					Quota_DestZ	:= Quota_PostZ + 						(* Quota Y Postazione *)
									Offset_Postazione_Z +				(* Offset Postazione *)	
									//Pallet_DimZ +						(* Dimensione/2 del Pallet/Cassa/Cavallina *)
									//Ojo formaciones en plano la altura de la base viene calculada en la  estructura
									// Forming
									Offset_Pallet_Z_90 + 				(* Offset Deposito Direzione Z del pallet *)
									Quota_FormaturaZ;					(* Quota di deposito Z da Formatura *)
										
					Quota_DestJ	:= Quota_FormaturaJ +					(* Quota di deposito Z da Formatura *)
									Offset_Pallet_J_90;					(* Offset Deposito inclinazione J del pallet *)
				
					(* Se ho l'abilitazione dell'utilizzo delle quote apprese,
						LE utilizzo come quote "buone" per eseguire il posizionamento *)				
					//Posizionamento lungo X
					//IF Apprendimento.X.Lato90.Stato = APPRENDIMENTO_ESEGUITO THEN
					//	Quota_DestX := Apprendimento.X.Lato90.QuotaRilevata;
					//END_IF
					////Posizionamento lungo Y lato 90°
					//IF Apprendimento.Y.Lato90.Stato = APPRENDIMENTO_ESEGUITO THEN
					//	Quota_DestY := Apprendimento.Y.Lato90.QuotaRilevata;
					//END_IF
					//Posizionamento lungo Z
					//Posizionamento lungo Z
					IF Apprendimento.Z.Lato90.Stato <> APPRENDIMENTO_DISABILITATO THEN
						IF Apprendimento.Z.Lato90.Stato = APPRENDIMENTO_ESEGUITO THEN
							Quota_ApproccioDestZ := Apprendimento.Z.Lato90.QuotaRilevata + Distanza_ApproccioFormaturaZ;
						ELSE
							Quota_ApproccioDestZ := Apprendimento.Z.Lato90.QuotaStart + Offset_Apprendimento_Z;
						END_IF
					ELSE
						Quota_ApproccioDestZ := Quota_DestZ +						(* Quota di deposito Z *)
												Distanza_ApproccioFormaturaZ;			(* Approccio Z da Formatura *)
					END_IF
					//Posizionamento lungo J lato 90°
					//IF Apprendimento.J.Lato90.Stato = APPRENDIMENTO_ESEGUITO THEN
					//	Quota_DestJ := Apprendimento.J.Lato90.QuotaRilevata;
					//END_IF			
				(*****************************************************************************************************************)
				(************************************************ QUOTE APPROCCIO ************************************************)
				(*****************************************************************************************************************)										
					Quota_ApproccioDestX	:= Quota_DestX;				(* Quota di deposito X *)
														
					Quota_ApproccioDestY 	:= Quota_DestY; 			(* Quota di deposito Y *)
											
					//Quota_ApproccioDestZ := Quota_DestZ +						(* Quota di deposito Z *)
					//						Distanza_ApproccioFormaturaZ;			(* Approccio Z da Formatura *)
										
					Quota_ApproccioDestJ	:= Quota_DestJ;				(* Quota di deposito J *)				
					
					
				END_IF
			{endregion}
			{Region "ANGOLO SX" }
			ANGOLO_SX :
				(*******************************************************************************************************************)
											(* Deposito su LASTRA con rotazione piano >90° e < 180°*)
				(*******************************************************************************************************************)
				IF Angolo_Destinazione > 90 THEN
					
					Quota_DestX	:= Quota_PostX + 						(* Quota X Postazione *)
									Offset_Postazione_X + 				(* Offset Postazione *)
									//Pallet_DimX/2 +						(* Dimensione/2 del Pallet/Cassa/Cavallina *)
									Offset_Pallet_X_180 +				(* Offset Deposito Direzione X del pallet *)
									Quota_FormaturaX;					(* Quota di deposito X da Formatura *)
				
					Quota_DestY := Quota_PostY + 						(* Quota Y Postazione *)
									IngombroDestinazioneY_Neg +
									Offset_Postazione_Y + 				(* Offset Postazione *)																							
									Pallet_DimY/2 +						(* Dimensione/2 del Pallet/Cassa/Cavallina *)
									Offset_Pallet_Y_180 +				(* Offset Deposito Direzione Y del pallet *)
									Quota_FormaturaY; 					(* Quota di deposito Y da Formatura *)
										
					Quota_DestZ	:= Quota_PostZ + 						(* Quota Y Postazione *)
									Offset_Postazione_Z +				(* Offset Postazione *)	
									//Pallet_DimZ +						(* Dimensione/2 del Pallet/Cassa/Cavallina *)
									Offset_Pallet_Z_180 + 				(* Offset Deposito Direzione Z del pallet *)
									(-ScostamentoVerticalePuntoCentrale) +		(* Sporgenza rispetto al filo pinza quando è in orizzontale *)
									Quota_FormaturaZ;					(* Quota di deposito Z da Formatura *)
							
					Quota_DestJ	:= Quota_FormaturaJ +					(* Quota di deposito Z da Formatura *)
									Offset_Pallet_J_180;				(* Offset Deposito inclinazione J del pallet *)
									
					(* Se ho l'abilitazione dell'utilizzo delle quote apprese,
						LE utilizzo come quote "buone" per eseguire il posizionamento *)				
					//Posizionamento lungo X
					IF Apprendimento.X.Lato180.Stato = APPRENDIMENTO_ESEGUITO THEN
						Quota_DestX := Apprendimento.X.Lato180.QuotaRilevata;
					END_IF
					//Posizionamento lungo Y lato 180°
					IF Apprendimento.Y.Lato180.Stato = APPRENDIMENTO_ESEGUITO THEN
						Quota_DestY := Apprendimento.Y.Lato180.QuotaRilevata;
					END_IF
					//Posizionamento lungo Z
					IF Apprendimento.Z.Lato180.Stato = APPRENDIMENTO_ESEGUITO THEN
						Quota_DestZ := Apprendimento.Z.Lato180.QuotaRilevata;
					END_IF
					//Posizionamento lungo J lato 180°
					IF Apprendimento.J.Lato180.Stato = APPRENDIMENTO_ESEGUITO THEN
						Quota_DestJ := Apprendimento.J.Lato180.QuotaRilevata;
					END_IF
				(*****************************************************************************************************************)
				(************************************************ QUOTE APPROCCIO ************************************************)
				(*****************************************************************************************************************)	
					
					(* Valutazione della Direzione dell'Asse X*)
					IF PosizioneAttuale_X >= Quota_DestX THEN // La posizione attuale è maggiore della posizione di destinazione 
						Quota_ApproccioDestX := Quota_DestX +					(* Quota di deposito X *)
												Distanza_ApproccioFormaturaX;		(* Approccio X da Formatura *)	
					ELSE // La posizione attuale è minore della posizione di destinazione 
						Quota_ApproccioDestX := Quota_DestX -					(* Quota di deposito X *)
												Distanza_ApproccioFormaturaX;		(* Approccio X da Formatura *)
					END_IF			
				
					Quota_ApproccioDestY := Quota_DestY + 						(* Quota di deposito Y *)
											Distanza_ApproccioFormaturaY; 			(* Approccio Y da Formatura *)
										
					Quota_ApproccioDestZ := Quota_DestZ +						(* Quota di deposito Z da Formatura *)
											Distanza_ApproccioFormaturaZ;			(* Approccio Z da Formatura *)
							
					Quota_ApproccioDestJ := Quota_DestJ +						(* Quota di deposito J da Forma*)	
											Distanza_ApproccioFormaturaJ;			(* Approccio J da Formatura *)
				(*******************************************************************************************************************)						
											(* Deposito su LASTRA con rotazione piano < 90° e >0°*)	
				(*******************************************************************************************************************)							
				ELSIF Angolo_Destinazione < 90 THEN
					
					Quota_DestX	:= Quota_PostX + 						(* Quota X Postazione *)
									Offset_Postazione_X + 				(* Offset Postazione *)
									//Pallet_DimX/2 +						(* Dimensione/2 del Pallet/Cassa/Cavallina *)
									Offset_Pallet_X_0 +					(* Offset Deposito Direzione X del pallet *)
									Quota_FormaturaX;					(* Quota di deposito X da Formatura *)
				
					Quota_DestY := Quota_PostY - 						(* Quota Y Postazione *)
									IngombroDestinazioneY_Pos +
									Offset_Postazione_Y + 				(* Offset Postazione *)																								
									Pallet_DimY/2 +						(* Dimensione/2 del Pallet/Cassa/Cavallina *)
									Offset_Pallet_Y_0 -					(* Offset Deposito Direzione Y del pallet *)
									Quota_FormaturaY; 					(* Quota di deposito Y da Formatura *)
										
					Quota_DestZ	:= Quota_PostZ + 						(* Quota Y Postazione *)
									Offset_Postazione_Z +				(* Offset Postazione *)	
									//Pallet_DimZ +						(* Dimensione/2 del Pallet/Cassa/Cavallina *)
									Offset_Pallet_Z_0 + 				(* Offset Deposito Direzione Z del pallet *)
									(-ScostamentoVerticalePuntoCentrale) +		(* Sporgenza rispetto al filo pinza quando è in orizzontale *)
									Quota_FormaturaZ;					(* Quota di deposito Z da Formatura *)
							
					Quota_DestJ	:= Quota_FormaturaJ +					(* Quota di deposito Z da Formatura *)
									Offset_Pallet_J_0;					(* Offset Deposito inclinazione J del pallet *)
									
					(* Se ho l'abilitazione dell'utilizzo delle quote apprese,
						LE utilizzo come quote "buone" per eseguire il posizionamento *)				
					//Posizionamento lungo X
					IF Apprendimento.X.Lato0.Stato = APPRENDIMENTO_ESEGUITO THEN
						Quota_DestX := Apprendimento.X.Lato0.QuotaRilevata;
					END_IF
					//Posizionamento lungo Y lato 0°
					IF Apprendimento.Y.Lato0.Stato = APPRENDIMENTO_ESEGUITO THEN
						Quota_DestY := Apprendimento.Y.Lato0.QuotaRilevata;
					END_IF
					//Posizionamento lungo Z
					IF Apprendimento.Z.Lato0.Stato = APPRENDIMENTO_ESEGUITO THEN
						Quota_DestZ := Apprendimento.Z.Lato0.QuotaRilevata;
					END_IF
					//Posizionamento lungo J lato 0°
					IF Apprendimento.J.Lato0.Stato = APPRENDIMENTO_ESEGUITO THEN
						Quota_DestJ := Apprendimento.J.Lato0.QuotaRilevata;
					END_IF
				(*****************************************************************************************************************)
				(************************************************ QUOTE APPROCCIO ************************************************)
				(*****************************************************************************************************************)	
					
					(* Valutazione della Direzione dell'Asse X*)
					IF PosizioneAttuale_X >= Quota_DestX THEN // La posizione attuale è maggiore della posizione di destinazione 
						Quota_ApproccioDestX := Quota_DestX +					(* Quota di deposito X *)
												Distanza_ApproccioFormaturaX;		(* Approccio X da Formatura *)	
					ELSE // La posizione attuale è minore della posizione di destinazione 
						Quota_ApproccioDestX := Quota_DestX -					(* Quota di deposito X *)
												Distanza_ApproccioFormaturaX;		(* Approccio X da Formatura *)
					END_IF			
				
					Quota_ApproccioDestY := Quota_DestY - 						(* Quota di deposito Y *)
											Distanza_ApproccioFormaturaY; 			(* Approccio Y da Formatura *)
										
					Quota_ApproccioDestZ := Quota_DestZ +						(* Quota di deposito Z *)
											Distanza_ApproccioFormaturaZ;			(* Approccio Z da Formatura *)
							
					Quota_ApproccioDestJ := Quota_DestJ +						(* Quota di deposito J *)
											Distanza_ApproccioFormaturaJ;			(* Approccio J da Formatura *)
							
				(*******************************************************************************************************************)						
											(* Deposito su LASTRA in cassa con rotazione piano = 90° *)
				(*******************************************************************************************************************)
				ELSE
					
					Quota_DestX	:= Quota_PostX + 						(* Quota X Postazione *)
									Offset_Postazione_X + 				(* Offset Postazione *)
									Pallet_DimX/2 +						(* Dimensione/2 del Pallet/Cassa/Cavallina *)
									Offset_Pallet_X_90;// +				(* Offset Deposito Direzione X del pallet *)
									//Quota_FormaturaX;					(* Quota di deposito X da Formatura *)
										
					Quota_DestY := Quota_PostY + 						(* Quota Y Postazione *)
									Offset_Postazione_Y + 				(* Offset Postazione *)																							
									Pallet_DimY/2 +						(* Dimensione/2 del Pallet/Cassa/Cavallina *)
									Offset_Pallet_Y_90;// +				(* Offset Deposito Direzione Y del pallet *)
									//Quota_FormaturaY; 					(* Quota di deposito Y da Formatura *)
											
					Quota_DestZ	:= Quota_PostZ + 						(* Quota Y Postazione *)
									Offset_Postazione_Z +				(* Offset Postazione *)	
									//Pallet_DimZ +						(* Dimensione/2 del Pallet/Cassa/Cavallina *)
									Offset_Pallet_Z_90 + 				(* Offset Deposito Direzione Z del pallet *)
									Quota_FormaturaZ;					(* Quota di deposito Z da Formatura *)
										
					Quota_DestJ	:= Quota_FormaturaJ;// +					(* Quota di deposito Z da Formatura *)
									//Offset_Pallet_J_90;					(* Offset Deposito inclinazione J del pallet *)
									
					(* Se ho l'abilitazione dell'utilizzo delle quote apprese,
						LE utilizzo come quote "buone" per eseguire il posizionamento *)				
					//Posizionamento lungo X
					IF Apprendimento.X.Lato90.Stato = APPRENDIMENTO_ESEGUITO THEN
						Quota_DestX := Apprendimento.X.Lato90.QuotaRilevata;
					END_IF
					//Posizionamento lungo Y lato 90°
					IF Apprendimento.Y.Lato90.Stato = APPRENDIMENTO_ESEGUITO THEN
						Quota_DestY := Apprendimento.Y.Lato90.QuotaRilevata;
					END_IF
					//Posizionamento lungo Z
					//IF Apprendimento.Z.Lato90.Stato = APPRENDIMENTO_ESEGUITO THEN
					//	Quota_DestZ := Apprendimento.Z.Lato90.QuotaRilevata + Offset_Apprendimento_Z;
					//ELSE
					//	Quota_DestZ := Apprendimento.Z.Lato90.QuotaStart;
					//END_IF
					//Posizionamento lungo Z
					IF Apprendimento.Z.Lato90.Stato <> APPRENDIMENTO_DISABILITATO THEN
						IF Apprendimento.Z.Lato90.Stato = APPRENDIMENTO_ESEGUITO THEN
							Quota_ApproccioDestZ := Apprendimento.Z.Lato90.QuotaRilevata + Distanza_ApproccioFormaturaZ;
						ELSE
							Quota_ApproccioDestZ := Apprendimento.Z.Lato90.QuotaStart + Offset_Apprendimento_Z;
						END_IF
					ELSE
						Quota_ApproccioDestZ := Quota_DestZ +						(* Quota di deposito Z *)
												Distanza_ApproccioFormaturaZ;			(* Approccio Z da Formatura *)
					END_IF		  
										
					//Posizionamento lungo J lato 90°
					IF Apprendimento.J.Lato90.Stato = APPRENDIMENTO_ESEGUITO THEN
						Quota_DestJ := Apprendimento.J.Lato90.QuotaRilevata;
					END_IF
							
				(*****************************************************************************************************************)
				(************************************************ QUOTE APPROCCIO ************************************************)
				(*****************************************************************************************************************)										
					Quota_ApproccioDestX	:= Quota_DestX;				(* Quota di deposito X *)
														
					Quota_ApproccioDestY 	:= Quota_DestY; 			(* Quota di deposito Y *)
											
					////Quota_ApproccioDestZ := Quota_DestZ +						(* Quota di deposito Z *)
					//						Distanza_ApproccioFormaturaZ;			(* Approccio Z da Formatura *)
										
					Quota_ApproccioDestJ	:= Quota_DestJ;				(* Quota di deposito J *)				
					
				END_IF
			{endregion}
			{Region "XDX_YCENTRALE" }
			XDX_YCENTRALE:
				(*******************************************************************************************************************)
											(* Deposito su LASTRA con rotazione piano >90° e < 180°*)
				(*******************************************************************************************************************)																		
				IF Angolo_Destinazione > 90 THEN
					
					Quota_DestX	:= Quota_PostX + 						(* Quota X Postazione *)
									Offset_Postazione_X - 				(* Offset Postazione *)
									Pallet_DimX/2 +						(* Dimensione/2 del Pallet/Cassa/Cavallina *)
									Offset_Pallet_X_180 +				(* Offset Deposito Direzione X del pallet *)
									Quota_FormaturaX;					(* Quota di deposito X da Formatura *)
				
					Quota_DestY := Quota_PostY + 						(* Quota Y Postazione *)
									Offset_Postazione_Y + 				(* Offset Postazione *)																								
									Pallet_DimY/2 -						(* Dimensione/2 del Pallet/Cassa/Cavallina *)
									//Offset_Pallet_Y_180 +				(* Offset Deposito Direzione Y del pallet *)
									Quota_FormaturaY; 					(* Quota di deposito Y da Formatura *)
										
					Quota_DestZ	:= Quota_PostZ + 						(* Quota Y Postazione *)
									Offset_Postazione_Z +				(* Offset Postazione *)	
									Pallet_DimZ +						(* Dimensione/2 del Pallet/Cassa/Cavallina *)
									Offset_Pallet_Z_180 + 				(* Offset Deposito Direzione Z del pallet *)
									Quota_FormaturaZ;					(* Quota di deposito Z da Formatura *)
							
					Quota_DestJ	:= Quota_FormaturaJ +					(* Quota di deposito Z da Formatura *)
									Offset_Pallet_J_180;				(* Offset Deposito inclinazione J del pallet *)
									
					(* Se ho l'abilitazione dell'utilizzo delle quote apprese,
						LE utilizzo come quote "buone" per eseguire il posizionamento *)				
					//Posizionamento lungo X
					IF Apprendimento.X.Lato180.Stato = APPRENDIMENTO_ESEGUITO THEN
						Quota_DestX := Apprendimento.X.Lato180.QuotaRilevata;
					END_IF
					//Posizionamento lungo Y lato 180°
					//IF Apprendimento.Y.Lato180.Stato = APPRENDIMENTO_ESEGUITO THEN
					//	Quota_DestY := Apprendimento.Y.Lato180.QuotaRilevata;
					//END_IF
					//Posizionamento lungo Z
					IF Apprendimento.Z.Lato180.Stato = APPRENDIMENTO_ESEGUITO THEN
						Quota_DestZ := Apprendimento.Z.Lato180.QuotaRilevata;
					END_IF
					//Posizionamento lungo J lato 180°
					IF Apprendimento.J.Lato180.Stato = APPRENDIMENTO_ESEGUITO THEN
						Quota_DestJ := Apprendimento.J.Lato180.QuotaRilevata;
					END_IF
									
				(*****************************************************************************************************************)
				(************************************************ QUOTE APPROCCIO ************************************************)
				(*****************************************************************************************************************)	
					Quota_ApproccioDestX	:= Quota_DestX;				(* Quota di deposito X *)
					//Quota_ApproccioDestY 	:= Quota_DestY; 			(* Quota di deposito Y *)
					IF CicloDiPrelievo THEN
						IF Apprendimento.Y.Lato90.Stato = APPRENDIMENTO_ESEGUITO THEN
							Quota_ApproccioDestY := Apprendimento.Y.Lato90.QuotaRilevata +	(* Quota rilevata Z *)
													Distanza_ApproccioFormaturaY;			(* Approccio Z da Formatura *)				
						ELSIF Apprendimento.Y.Lato90.Stato <> APPRENDIMENTO_ESEGUITO THEN
							Quota_ApproccioDestY := Quota_DestY + 						(* Quota di deposito Y *)
													Distanza_ApproccioFormaturaY+ 			(* Approccio Y da Formatura *)
													Offset_Apprendimento_Y;							
						END_IF
					ELSE
						//Posizionamento lungo Z lato 90°
						IF Apprendimento.Y.Lato90.Stato = APPRENDIMENTO_ESEGUITO THEN
							Quota_DestY := Apprendimento.Y.Lato90.QuotaRilevata +
											Distanza_ApproccioFormaturaY;
						END_IF
					END_IF
					
					Quota_ApproccioDestZ := Quota_DestZ +						(* Quota di deposito Z *)
											Distanza_ApproccioFormaturaZ;			(* Approccio Z da Formatura *)
										
					Quota_ApproccioDestJ	:= Quota_DestJ;				(* Quota di deposito J *)				
									
				(*******************************************************************************************************************)						
											(* Deposito su LASTRA con rotazione piano < 90° e >0°*)	
				(*******************************************************************************************************************)							
				ELSIF Angolo_Destinazione < 90 THEN
					
					Quota_DestX	:= Quota_PostX + 						(* Quota X Postazione *)
									Offset_Postazione_X - 				(* Offset Postazione *)
									Pallet_DimX/2 +						(* Dimensione/2 del Pallet/Cassa/Cavallina *)
									Offset_Pallet_X_0 +					(* Offset Deposito Direzione X del pallet *)
									Quota_FormaturaX;					(* Quota di deposito X da Formatura *)
				
					Quota_DestY := Quota_PostY - 						(* Quota Y Postazione *)
									Offset_Postazione_Y - 				(* Offset Postazione *)																							
									Pallet_DimY/2 -						(* Dimensione/2 del Pallet/Cassa/Cavallina *)
									//Offset_Pallet_Y_0 +					(* Offset Deposito Direzione Y del pallet *)
									Quota_FormaturaY; 					(* Quota di deposito Y da Formatura *)
										
					Quota_DestZ	:= Quota_PostZ + 						(* Quota Y Postazione *)
									Offset_Postazione_Z +				(* Offset Postazione *)	
									Pallet_DimZ +						(* Dimensione/2 del Pallet/Cassa/Cavallina *)
									Offset_Pallet_Z_0 + 				(* Offset Deposito Direzione Z del pallet *)
									Quota_FormaturaZ;					(* Quota di deposito Z da Formatura *)
							
					Quota_DestJ	:= Quota_FormaturaJ +					(* Quota di deposito Z da Formatura *)
									Offset_Pallet_J_0;					(* Offset Deposito inclinazione J del pallet *)
									
					(* Se ho l'abilitazione dell'utilizzo delle quote apprese,
						LE utilizzo come quote "buone" per eseguire il posizionamento *)				
					//Posizionamento lungo X
					IF Apprendimento.X.Lato0.Stato = APPRENDIMENTO_ESEGUITO THEN
						Quota_DestX := Apprendimento.X.Lato0.QuotaRilevata;
					END_IF
					//Posizionamento lungo Y lato 0°
					//IF Apprendimento.Y.Lato0.Stato = APPRENDIMENTO_ESEGUITO THEN
					//	Quota_DestY := Apprendimento.Y.Lato0.QuotaRilevata;
					//END_IF
					IF CicloDiPrelievo THEN
						IF Apprendimento.Y.Lato90.Stato = APPRENDIMENTO_ESEGUITO THEN
							Quota_ApproccioDestY := Apprendimento.Y.Lato90.QuotaRilevata -	(* Quota rilevata Z *)
													Distanza_ApproccioFormaturaY;			(* Approccio Z da Formatura *)				
						ELSIF Apprendimento.Y.Lato90.Stato <> APPRENDIMENTO_ESEGUITO THEN
							Quota_ApproccioDestY := Quota_DestY - 						(* Quota di deposito Y *)
													Distanza_ApproccioFormaturaY- 			(* Approccio Y da Formatura *)
													Offset_Apprendimento_Y;							
						END_IF
					ELSE
						//Posizionamento lungo Z lato 90°
						IF Apprendimento.Y.Lato90.Stato = APPRENDIMENTO_ESEGUITO THEN
							Quota_DestY := Apprendimento.Y.Lato90.QuotaRilevata -
											Distanza_ApproccioFormaturaY;
						END_IF
					END_IF
					//Posizionamento lungo Z
					IF Apprendimento.Z.Lato0.Stato = APPRENDIMENTO_ESEGUITO THEN
						Quota_DestZ := Apprendimento.Z.Lato0.QuotaRilevata;
					END_IF
					//Posizionamento lungo J lato 0°
					IF Apprendimento.J.Lato0.Stato = APPRENDIMENTO_ESEGUITO THEN
						Quota_DestJ := Apprendimento.J.Lato0.QuotaRilevata;
					END_IF
									
				(*****************************************************************************************************************)
				(************************************************ QUOTE APPROCCIO ************************************************)
				(*****************************************************************************************************************)	
					
					(* Valutazione della Direzione dell'Asse X*)
					IF PosizioneAttuale_X >= Quota_DestX THEN // La posizione attuale è maggiore della posizione di destinazione 
						Quota_ApproccioDestX := Quota_DestX +					(* Quota di deposito X *)
												Distanza_ApproccioFormaturaX;		(* Approccio X da Formatura *)	
					ELSE // La posizione attuale è minore della posizione di destinazione 
						Quota_ApproccioDestX := Quota_DestX -					(* Quota di deposito X *)
												Distanza_ApproccioFormaturaX;		(* Approccio X da Formatura *)
					END_IF			
				
					Quota_ApproccioDestY := Quota_DestY - 						(* Quota di deposito Y *)
											Distanza_ApproccioFormaturaY; 			(* Approccio Y da Formatura *)
										
					Quota_ApproccioDestZ := Quota_DestZ +						(* Quota di deposito Z *)
											Distanza_ApproccioFormaturaZ;			(* Approccio Z da Formatura *)
							
					Quota_ApproccioDestJ := Quota_DestJ +						(* Quota di deposito J *)
											Distanza_ApproccioFormaturaJ;			(* Approccio J da Formatura *)				
							
				(*******************************************************************************************************************)						
											(* Deposito su LASTRA in cassa con rotazione piano = 90° *)
				(*******************************************************************************************************************)
				ELSE
					
					Quota_DestX	:= Quota_PostX + 						(* Quota X Postazione *)
									Offset_Postazione_X - 				(* Offset Postazione *)
									Pallet_DimX/2 +						(* Dimensione/2 del Pallet/Cassa/Cavallina *)
									Offset_Pallet_X_90 +				(* Offset Deposito Direzione X del pallet *)
									Quota_FormaturaX;					(* Quota di deposito X da Formatura *)
														
					Quota_DestY := Quota_PostY + 						(* Quota Y Postazione *)
									Offset_Postazione_Y + 				(* Offset Postazione *)																							
									//Pallet_DimY/2 +						(* Dimensione/2 del Pallet/Cassa/Cavallina *)
									//Offset_Pallet_Y_90 +				(* Offset Deposito Direzione Y del pallet *)
									Quota_FormaturaY; 					(* Quota di deposito Y da Formatura *)
											
					Quota_DestZ	:= Quota_PostZ + 						(* Quota Y Postazione *)
									Offset_Postazione_Z +				(* Offset Postazione *)	
									Pallet_DimZ +						(* Dimensione/2 del Pallet/Cassa/Cavallina *)
									Offset_Pallet_Z_90 + 				(* Offset Deposito Direzione Z del pallet *)
									Quota_FormaturaZ;					(* Quota di deposito Z da Formatura *)
										
					Quota_DestJ	:= Quota_FormaturaJ +					(* Quota di deposito Z da Formatura *)
									Offset_Pallet_J_90;					(* Offset Deposito inclinazione J del pallet *)
					
					(* Se ho l'abilitazione dell'utilizzo delle quote apprese,
						LE utilizzo come quote "buone" per eseguire il posizionamento *)				
					//Posizionamento lungo X
					IF Apprendimento.X.Lato90.Stato = APPRENDIMENTO_ESEGUITO THEN
						Quota_DestX := Apprendimento.X.Lato90.QuotaRilevata;
					END_IF
					//Posizionamento lungo Y lato 90°
					IF Apprendimento.Y.Lato90.Stato = APPRENDIMENTO_ESEGUITO THEN
						Quota_DestY := Apprendimento.Y.Lato90.QuotaRilevata;
					END_IF
					//Posizionamento lungo Z
					IF CicloDiPrelievo THEN
						IF Apprendimento.Z.Lato90.Stato = APPRENDIMENTO_ESEGUITO THEN
							Quota_ApproccioDestZ := Apprendimento.Z.Lato90.QuotaRilevata +	(* Quota rilevata Z *)
													Distanza_ApproccioFormaturaZ;			(* Approccio Z da Formatura *)				
						ELSIF Apprendimento.Z.Lato90.Stato <> APPRENDIMENTO_ESEGUITO THEN
							Quota_ApproccioDestZ := Quota_PostZ + 						(* Quota Y Postazione *)
													Offset_Postazione_Z +				(* Offset Postazione *)	
													Offset_Pallet_Z_0 +					(* Offset Direzione Z del pall*)
													HmaxElemento +						(* Quota di deposito Z *)
													Offset_Apprendimento_Z;							
						END_IF
					ELSE
						//Posizionamento lungo Z lato 90°
						IF Apprendimento.Z.Lato90.Stato = APPRENDIMENTO_ESEGUITO THEN
							Quota_DestZ := Apprendimento.Z.Lato90.QuotaRilevata;
						END_IF
						Quota_ApproccioDestZ := Quota_DestZ +						(* Quota di deposito Z *)
												Distanza_ApproccioFormaturaZ;			(* Approccio Z da Formatura *)
					END_IF
					//Posizionamento lungo J lato 90°
					IF Apprendimento.J.Lato90.Stato = APPRENDIMENTO_ESEGUITO THEN
						Quota_DestJ := Apprendimento.J.Lato90.QuotaRilevata;
					END_IF
									
				(*****************************************************************************************************************)
				(************************************************ QUOTE APPROCCIO ************************************************)
				(*****************************************************************************************************************)										
					Quota_ApproccioDestX	:= Quota_DestX;				(* Quota di deposito X *)
														
					Quota_ApproccioDestY 	:= Quota_DestY; 			(* Quota di deposito Y *)
											
					//Quota_ApproccioDestZ := Quota_DestZ +						(* Quota di deposito Z *)
					//						Distanza_ApproccioFormaturaZ;			(* Approccio Z da Formatura *)
										
					Quota_ApproccioDestJ	:= Quota_DestJ;				(* Quota di deposito J *)				
				END_IF
			{endregion}
			{Region "XSX_YCENTRALE" }
			XSX_YCENTRALE:
				(*******************************************************************************************************************)
											(* Deposito su LASTRA con rotazione piano >90° e < 180°*)
				(*******************************************************************************************************************)
				IF Angolo_Destinazione > 90 THEN
					
					Quota_DestX	:= Quota_PostX + 						(* Quota X Postazione *)
									Offset_Postazione_X + 				(* Offset Postazione *)
									Pallet_DimX/2 +						(* Dimensione/2 del Pallet/Cassa/Cavallina *)
									Offset_Pallet_X_180 +				(* Offset Deposito Direzione X del pallet *)
									Quota_FormaturaX;					(* Quota di deposito X da Formatura *)
				
					Quota_DestY := Quota_PostY + 						(* Quota Y Postazione *)
									Offset_Postazione_Y + 				(* Offset Postazione *)																							
									//Pallet_DimY/2 +						(* Dimensione/2 del Pallet/Cassa/Cavallina *)
									//Offset_Pallet_Y_180 +				(* Offset Deposito Direzione Y del pallet *)
									Quota_FormaturaY; 					(* Quota di deposito Y da Formatura *)
										
					Quota_DestZ	:= Quota_PostZ + 						(* Quota Y Postazione *)
									Offset_Postazione_Z +				(* Offset Postazione *)	
									Pallet_DimZ +						(* Dimensione/2 del Pallet/Cassa/Cavallina *)
									Offset_Pallet_Z_180 + 				(* Offset Deposito Direzione Z del pallet *)
									Quota_FormaturaZ;					(* Quota di deposito Z da Formatura *)
							
					Quota_DestJ	:= Quota_FormaturaJ +					(* Quota di deposito Z da Formatura *)
									Offset_Pallet_J_180;				(* Offset Deposito inclinazione J del pallet *)
									
					(* Se ho l'abilitazione dell'utilizzo delle quote apprese,
						LE utilizzo come quote "buone" per eseguire il posizionamento *)				
					//Posizionamento lungo X
					IF Apprendimento.X.Lato180.Stato = APPRENDIMENTO_ESEGUITO THEN
						Quota_DestX := Apprendimento.X.Lato180.QuotaRilevata;
					END_IF
					//Posizionamento lungo Y lato 180°
					IF Apprendimento.Y.Lato180.Stato = APPRENDIMENTO_ESEGUITO THEN
						Quota_DestY := Apprendimento.Y.Lato180.QuotaRilevata;
					END_IF
					//Posizionamento lungo Z
					IF Apprendimento.Z.Lato180.Stato = APPRENDIMENTO_ESEGUITO THEN
						Quota_DestZ := Apprendimento.Z.Lato180.QuotaRilevata;
					END_IF
					//Posizionamento lungo J lato 180°
					IF Apprendimento.J.Lato180.Stato = APPRENDIMENTO_ESEGUITO THEN
						Quota_DestJ := Apprendimento.J.Lato180.QuotaRilevata;
					END_IF				
					
				(*****************************************************************************************************************)
				(************************************************ QUOTE APPROCCIO ************************************************)
				(*****************************************************************************************************************)	
					
					(* Valutazione della Direzione dell'Asse X*)
					IF PosizioneAttuale_X >= Quota_DestX THEN // La posizione attuale è maggiore della posizione di destinazione 
						Quota_ApproccioDestX := Quota_DestX +					(* Quota di deposito X *)
												Distanza_ApproccioFormaturaX;		(* Approccio X da Formatura *)	
					ELSE // La posizione attuale è minore della posizione di destinazione 
						Quota_ApproccioDestX := Quota_DestX -					(* Quota di deposito X *)
												Distanza_ApproccioFormaturaX;		(* Approccio X da Formatura *)
					END_IF			
				
					Quota_ApproccioDestY := Quota_DestY + 						(* Quota di deposito Y *)
											Distanza_ApproccioFormaturaY; 			(* Approccio Y da Formatura *)
										
					Quota_ApproccioDestZ := Quota_DestZ +						(* Quota di deposito Z da Formatura *)
											Distanza_ApproccioFormaturaZ;			(* Approccio Z da Formatura *)
							
					Quota_ApproccioDestJ := Quota_DestJ +						(* Quota di deposito J da Forma*)	
											Distanza_ApproccioFormaturaJ;			(* Approccio J da Formatura *)
				(*******************************************************************************************************************)						
											(* Deposito su LASTRA con rotazione piano < 90° e >0°*)	
				(*******************************************************************************************************************)							
				ELSIF Angolo_Destinazione < 90 THEN
					
					Quota_DestX	:= Quota_PostX + 						(* Quota X Postazione *)
									Offset_Postazione_X + 				(* Offset Postazione *)
									Pallet_DimX/2 +						(* Dimensione/2 del Pallet/Cassa/Cavallina *)
									Offset_Pallet_X_0 +					(* Offset Deposito Direzione X del pallet *)
									Quota_FormaturaX;					(* Quota di deposito X da Formatura *)
				
					Quota_DestY := Quota_PostY + 						(* Quota Y Postazione *)
									Offset_Postazione_Y + 				(* Offset Postazione *)																								
									//Pallet_DimY/2 -						(* Dimensione/2 del Pallet/Cassa/Cavallina *)
									//Offset_Pallet_Y_0 +					(* Offset Deposito Direzione Y del pallet *)
									Quota_FormaturaY; 					(* Quota di deposito Y da Formatura *)
										
					Quota_DestZ	:= Quota_PostZ + 						(* Quota Y Postazione *)
									Offset_Postazione_Z +				(* Offset Postazione *)	
									Pallet_DimZ +						(* Dimensione/2 del Pallet/Cassa/Cavallina *)
									Offset_Pallet_Z_90 + 				(* Offset Deposito Direzione Z del pallet *)
									Quota_FormaturaZ;					(* Quota di deposito Z da Formatura *)
							
					Quota_DestJ	:= Quota_FormaturaJ +					(* Quota di deposito Z da Formatura *)
									Offset_Pallet_J_0;					(* Offset Deposito inclinazione J del pallet *)
									
					(* Se ho l'abilitazione dell'utilizzo delle quote apprese,
						LE utilizzo come quote "buone" per eseguire il posizionamento *)				
					//Posizionamento lungo X
					IF Apprendimento.X.Lato0.Stato = APPRENDIMENTO_ESEGUITO THEN
						Quota_DestX := Apprendimento.X.Lato0.QuotaRilevata;
					END_IF
					//Posizionamento lungo Y lato 0°
					IF Apprendimento.Y.Lato0.Stato = APPRENDIMENTO_ESEGUITO THEN
						Quota_DestY := Apprendimento.Y.Lato0.QuotaRilevata;
					END_IF
					//Posizionamento lungo Z
					IF Apprendimento.Z.Lato0.Stato = APPRENDIMENTO_ESEGUITO THEN
						Quota_DestZ := Apprendimento.Z.Lato0.QuotaRilevata;
					END_IF
					//Posizionamento lungo J lato 0°
					IF Apprendimento.J.Lato0.Stato = APPRENDIMENTO_ESEGUITO THEN
						Quota_DestJ := Apprendimento.J.Lato0.QuotaRilevata;
					END_IF		
					
				(*****************************************************************************************************************)
				(************************************************ QUOTE APPROCCIO ************************************************)
				(*****************************************************************************************************************)	
					
					(* Valutazione della Direzione dell'Asse X*)
					IF PosizioneAttuale_X >= Quota_DestX THEN // La posizione attuale è maggiore della posizione di destinazione 
						Quota_ApproccioDestX := Quota_DestX +					(* Quota di deposito X *)
												Distanza_ApproccioFormaturaX;		(* Approccio X da Formatura *)	
					ELSE // La posizione attuale è minore della posizione di destinazione 
						Quota_ApproccioDestX := Quota_DestX -					(* Quota di deposito X *)
												Distanza_ApproccioFormaturaX;		(* Approccio X da Formatura *)
					END_IF			
				
					Quota_ApproccioDestY := Quota_DestY - 						(* Quota di deposito Y *)
											Distanza_ApproccioFormaturaY; 			(* Approccio Y da Formatura *)
										
					Quota_ApproccioDestZ := Quota_DestZ +						(* Quota di deposito Z *)
											Distanza_ApproccioFormaturaZ;			(* Approccio Z da Formatura *)
							
					Quota_ApproccioDestJ := Quota_DestJ +						(* Quota di deposito J *)
											Distanza_ApproccioFormaturaJ;			(* Approccio J da Formatura *)
							
				(*******************************************************************************************************************)						
											(* Deposito su LASTRA in cassa con rotazione piano = 90° *)
				(*******************************************************************************************************************)
				ELSE
					
					Quota_DestX	:= Quota_PostX + 						(* Quota X Postazione *)
									Offset_Postazione_X + 				(* Offset Postazione *)
									Pallet_DimX/2 +						(* Dimensione/2 del Pallet/Cassa/Cavallina *)
									Offset_Pallet_X_90 +				(* Offset Deposito Direzione X del pallet *)
									Quota_FormaturaX;					(* Quota di deposito X da Formatura *)
										
					Quota_DestY := Quota_PostY + 						(* Quota Y Postazione *)
									Offset_Postazione_Y + 				(* Offset Postazione *)																							
									//Pallet_DimY/2 +						(* Dimensione/2 del Pallet/Cassa/Cavallina *)
									//Offset_Pallet_Y_90 +				(* Offset Deposito Direzione Y del pallet *)
									Quota_FormaturaY; 					(* Quota di deposito Y da Formatura *)
											
					Quota_DestZ	:= Quota_PostZ + 						(* Quota Y Postazione *)
									Offset_Postazione_Z +				(* Offset Postazione *)	
									Pallet_DimZ +						(* Dimensione/2 del Pallet/Cassa/Cavallina *)
									Offset_Pallet_Z_90 + 				(* Offset Deposito Direzione Z del pallet *)
									Quota_FormaturaZ;					(* Quota di deposito Z da Formatura *)
										
					Quota_DestJ	:= Quota_FormaturaJ +					(* Quota di deposito Z da Formatura *)
									Offset_Pallet_J_90;					(* Offset Deposito inclinazione J del pallet *)
					
					(* Se ho l'abilitazione dell'utilizzo delle quote apprese,
						LE utilizzo come quote "buone" per eseguire il posizionamento *)				
					//Posizionamento lungo X
					IF Apprendimento.X.Lato0.Stato = APPRENDIMENTO_ESEGUITO THEN
						Quota_DestX := Apprendimento.X.Lato0.QuotaRilevata;
					END_IF
					//Posizionamento lungo Y lato 0°
					IF Apprendimento.Y.Lato0.Stato = APPRENDIMENTO_ESEGUITO THEN
						Quota_DestY := Apprendimento.Y.Lato0.QuotaRilevata;
					END_IF
					//Posizionamento lungo Z
					IF Apprendimento.Z.Lato0.Stato = APPRENDIMENTO_ESEGUITO THEN
						Quota_DestZ := Apprendimento.Z.Lato0.QuotaRilevata;
					END_IF
					//Posizionamento lungo J lato 0°
					IF Apprendimento.J.Lato0.Stato = APPRENDIMENTO_ESEGUITO THEN
						Quota_DestJ := Apprendimento.J.Lato0.QuotaRilevata;
					END_IF	
				(*****************************************************************************************************************)
				(************************************************ QUOTE APPROCCIO ************************************************)
				(*****************************************************************************************************************)										
					Quota_ApproccioDestX	:= Quota_DestX;				(* Quota di deposito X *)
														
					Quota_ApproccioDestY 	:= Quota_DestY; 			(* Quota di deposito Y *)
											
					Quota_ApproccioDestZ := Quota_DestZ +						(* Quota di deposito Z *)
											Distanza_ApproccioFormaturaZ;			(* Approccio Z da Formatura *)
										
					Quota_ApproccioDestJ	:= Quota_DestJ;				(* Quota di deposito J *)
					
				END_IF
			{endregion}		
							
		ELSE
			Errore.Code := ErrWAM_FTC_PostazioneNONDefinita;
		END_CASE
	{endregion}	
	ELSE
		Errore.Code := ErrGENERICO;		
END_CASE
{region " Gestione Approccio "}	
CASE TipologiaTraiettoria OF
	
	TRAIETTORIA_CON_APPROCCIO:
		RETURN;
	
	TRAIETTORIA_SENZA_APPROCCIO:
		(*****************************************************************************************************************)
		(************************************************ QUOTE APPROCCIO ************************************************)
		(*****************************************************************************************************************)										
		Quota_ApproccioDestX	:= Quota_DestX;				(* Quota di deposito X *)
											
		Quota_ApproccioDestY 	:= Quota_DestY; 			(* Quota di deposito Y *)
								
		Quota_ApproccioDestZ 	:= Quota_DestZ; 			(* Quota di deposito Z *)
							
		Quota_ApproccioDestJ	:= Quota_DestJ;				(* Quota di deposito J *)
		RETURN;	
END_CASE
{endregion}

END_FUNCTION_BLOCK

// ---- POUs/TFPalletizerData_Lastre/Formatura/Calcolo_Formatura_Completa.TcPOU
FUNCTION_BLOCK Calcolo_Formatura_Completa
VAR_INPUT
	
	Supporto : TFMachinePalletizer_Pallet;
	
	//Materiale : ARRAY [0..MAXTYPE_SLABLAYER] OF Type_SlabLayer;	// Tipo di materiale, Lastra, Falda e dimensioni
	Materiale 			: ARRAY [0..MAXTYPE_SLABLAYER] OF TFMachinePalletizer_PlaceElement;	// Tipo di materiale, Lastra, Falda e dimensioni
	TipoElementoDep 	: ARRAY [1..MAXFORMINGSLAB] OF e_Tipo_Elemento_Da_Lavorare;	// Tipologia del n-esimo elemento di Materiale da depositare (Lstra-falda-terminatore)
	DimensionesPiezasDifEsPiking	: ARRAY  [1..MAXELEMENTLIST] OF ES_dimensionPiezaLadoA_ladoB;
	TipoRisultato 		: UINT := 3;// Punto utilizzato per coordinate finali di deposito lastra/falda, 1 interno, 2 centro, 3 esterno(default)
	TipoOrdinamento 	: UINT := 1;//Tipologia di ordinamento in deposito 1= alternato (lastra DX-Lastra SX), 2 = consecutivo(prima un lato, poi l'altro lato), 3 = solo lato 0°, 4 = solo lato 180°
	NumeroElementiDaDepositare : UINT;
	
	
	PulisciMemoria 								: BOOL;
	CalcolaFormatura 							: BOOL;
	CalculoEstacionPickinPiezasDiferentes		: BOOL;
	HabiCalTodasCordenadas						: BOOL;
END_VAR

VAR_OUTPUT
	(* Variabili di uscita della posizione finale del punto di deposito della lastra/falda *)
	XFinale : ARRAY [1..MAXFORMINGSLAB] OF LREAL;		// Coordinata X punto finale n-esima lastra/falda depositata
	YFinale : ARRAY [1..MAXFORMINGSLAB] OF LREAL;		// Coordinata Y punto finale n-esima lastra/falda depositata
	ZFinale : ARRAY [1..MAXFORMINGSLAB] OF LREAL;		// Coordinata Z punto finale n-esima lastra/falda depositata
	JFinale : ARRAY [1..MAXFORMINGSLAB] OF LREAL;		// Coordinata J punto finale n-esima lastra/falda depositata
	
	XFinaleLado_0Grados : ARRAY [1..MAXFORMINGSLAB] OF LREAL;		// Coordinata X punto finale n-esima lastra/falda depositata
	YFinaleLado_0Grados : ARRAY [1..MAXFORMINGSLAB] OF LREAL;		// Coordinata Y punto finale n-esima lastra/falda depositata
	ZFinaleLado_0Grados : ARRAY [1..MAXFORMINGSLAB] OF LREAL;		// Coordinata Z punto finale n-esima lastra/falda depositata
	JFinaleLado_0Grados : ARRAY [1..MAXFORMINGSLAB] OF LREAL;		// Coordinata J punto finale n-esima lastra/falda depositata
	
	XFinaleLado_180Grados : ARRAY [1..MAXFORMINGSLAB] OF LREAL;		// Coordinata X punto finale n-esima lastra/falda depositata
	YFinaleLado_180Grados : ARRAY [1..MAXFORMINGSLAB] OF LREAL;		// Coordinata Y punto finale n-esima lastra/falda depositata
	ZFinaleLado_180Grados : ARRAY [1..MAXFORMINGSLAB] OF LREAL;		// Coordinata Z punto finale n-esima lastra/falda depositata
	JFinaleLado_180Grados : ARRAY [1..MAXFORMINGSLAB] OF LREAL;		// Coordinata J punto finale n-esima lastra/falda depositata
	
	CoorFinaleLado_Pri0_Des180 : ARRAY [1..MAXFORMINGSLAB] OF Es_CoordenadasCaballeteLadoA_ladoB ;		// Coordinata X punto finale n-esima lastra/falda depositata
	
	
	CoordenadasCaballete 				: ARRAY [1..MAXFORMINGSLAB] OF Es_CoordenadasCaballeteLadoA_ladoB ;
	
	FormingSlab 						: TFMachinePalletizer_FormingForSlab;
	PulisciMemoriaDone					: BOOL;
	CalcolaFormaturaDone 				: BOOL;
	Errore 								: UINT;
END_VAR

VAR_IN_OUT
	
END_VAR

VAR
	TipoDeposito : e_TipologiaDeposito;				// ORIZZONTALE O INCLINATO
	OrdineDepositoSxDx : ARRAY [1..MAXFORMINGSLAB] OF e_Tipo_Elemento_Da_Lavorare;	// Ordine deposito materiale per i due lati, sx e dx (considero di avere il medesimo ordine di deposito dai due lati) (CAVALLINA-INCLINATO)
	
	Spessore_Lastra_Inclinata 					: ARRAY [1..MAXFORMINGSLAB/2] OF LREAL;				// Occupazione in larghezza della singola lastra (CAVALLINA-INCLINATO)
	Spessore_Lastra_Inclinata_Cumulato 			: ARRAY [1..MAXFORMINGSLAB/2] OF LREAL;	// Occupazione in larghezza delle nlastre lastre cumulate (CAVALLINA)
	
	Spessore_Lastra_Inclinata_lado_A_B 			: ARRAY [1..MAXFORMINGSLAB/2] OF ES_SpesoreLastra_A_B;
	Spessore_Lastra_Inclinata_Cumulato_A_B 		: ARRAY [1..MAXFORMINGSLAB/2] OF ES_SpesoreLastra_A_B;
	
	
	Spessore_Lastra : ARRAY [1..MAXFORMINGSLAB] OF LREAL;							// Occupazione in altezza della singola lastra (CASSA-ORIZZONTALE)
	Spessore_Lastra_Cumulato : ARRAY [1..MAXFORMINGSLAB] OF LREAL;					// Occupazione in altezza delle nlastre lastre cumulate (CASSA-ORIZZONTALE)
	
	
	
	YCoordinataAppoggioLastra :  ARRAY [1..MAXFORMINGSLAB/2] OF LREAL;		// Coordinata Y del punto di appoggio della lastra sulla base della cavallina  (CAVALLINA-INCLINATO)
	ZCoordinataAppoggioLastra :  ARRAY [1..MAXFORMINGSLAB/2] OF LREAL;		// Coordinata Z del punto di appoggio della lastra sulla base della cavallina  (CAVALLINA-INCLINATO)
	
	YCoordinataAppoggioLastra_A_B :  ARRAY [1..MAXFORMINGSLAB/2] OF ES_SpesoreLastra_A_B;
	ZCoordinataAppoggioLastra_A_B :  ARRAY [1..MAXFORMINGSLAB/2] OF ES_SpesoreLastra_A_B;
	
	B 	: LREAL;	// Base della cavallina (include i due lati)  (CAVALLINA-INCLINATO)
	B2	: LREAL;	// Base della cavallina (include i due lati)  (CAVALLINA-INCLINATO)
	CorYIz  : LREAL;
	CorYDe : LREAL;
	TipoCalculo : UINT := 0;
	
	BaseAlgulo : LREAL ;
	b1 : LREAL;	// base del triangolo rettangolo dell'angolo alfa  (CAVALLINA-INCLINATO)
	h1 : LREAL; // altezza del triangolo rettangolo dell'angolo alfa  (CAVALLINA-INCLINATO)
	Yd1 : ARRAY [1..MAXFORMINGSLAB/2] OF LREAL;	// Spostamento Centro lastra da inizio lastra in Y  (CAVALLINA-INCLINATO)
	Zd1 : ARRAY [1..MAXFORMINGSLAB/2] OF LREAL;	// Spostamento Centro lastra da inizio lastra in Z  (CAVALLINA-INCLINATO)
	Yd2 : ARRAY [1..MAXFORMINGSLAB/2] OF LREAL;	// Spostamento Esterno lastra da inizio lastra in Y  (CAVALLINA-INCLINATO)
	Zd2 : ARRAY [1..MAXFORMINGSLAB/2] OF LREAL;	// Spostamento Esterno lastra da inizio lastra in Z  (CAVALLINA-INCLINATOCAVALLINA)
	Yd3 : ARRAY [1..MAXFORMINGSLAB/2] OF LREAL;	// Spostamento Y dovuto al lato inclinato base appoggio  (CAVALLINA-INCLINATO)
	Zd3 : ARRAY [1..MAXFORMINGSLAB/2] OF LREAL;	// Spostamento Z dovuto al lato inclinato base appoggio  (CAVALLINA-INCLINATO)
	CI : ARRAY [1..MAXFORMINGSLAB/2] OF LREAL;	// Proiezione mancante della lastra dovuta al piano inclinato (CI) - Valorizzata solo se Beta >0  (CAVALLINA-INCLINATO)
	
	Yd1_A_B : ARRAY [1..MAXFORMINGSLAB/2] OF ES_SpesoreLastra_A_B;	// Spostamento Centro lastra da inizio lastra in Y  (CAVALLINA-INCLINATO)
	Zd1_A_B : ARRAY [1..MAXFORMINGSLAB/2] OF ES_SpesoreLastra_A_B;	// Spostamento Centro lastra da inizio lastra in Z  (CAVALLINA-INCLINATO)
	Yd2_A_B : ARRAY [1..MAXFORMINGSLAB/2] OF ES_SpesoreLastra_A_B;	// Spostamento Esterno lastra da inizio lastra in Y  (CAVALLINA-INCLINATO)
	Zd2_A_B : ARRAY [1..MAXFORMINGSLAB/2] OF ES_SpesoreLastra_A_B;	// Spostamento Esterno lastra da inizio lastra in Z  (CAVALLINA-INCLINATOCAVALLINA)
	Yd3_A_B : ARRAY [1..MAXFORMINGSLAB/2] OF ES_SpesoreLastra_A_B;	// Spostamento Y dovuto al lato inclinato base appoggio  (CAVALLINA-INCLINATO)
	Zd3_A_B : ARRAY [1..MAXFORMINGSLAB/2] OF ES_SpesoreLastra_A_B;	// Spostamento Z dovuto al lato inclinato base appoggio  (CAVALLINA-INCLINATO)
	CI_A_B : ARRAY [1..MAXFORMINGSLAB/2] OF ES_SpesoreLastra_A_B;	// Proiezione mancante della lastra dovuta al piano inclinato (CI) - Valorizzata solo se Beta >0  (CAVALLINA-INCLINATO)
	
	
	
	rad90 : LREAL;		// 90° in radianti
	
	(* Angoli piani appoggio lastre, laterale (alfa) e base (beta) cavallina *)
	AngoloAlfa_rad : LREAL;		// Angolo superiore laterale appoggio della lastra (in radianti)  (CAVALLINA-INCLINATO)
	AlgoloAlfa_gradi : LREAL; 	// Angolo superiore laterale appoggio della lastra (in gradi)  (CAVALLINA-INCLINATO)
	AngoloBeta_rad : LREAL;		// Angolo del piano inclinato di appoggio della lastra in radianti  (CAVALLINA-INCLINATO)
	AngoloBeta_gradi : LREAL; 	// Angolo del piano inclinato di appoggio della lastra in gradi  (CAVALLINA-INCLINATO)
	
	QuotaYinizioLastra : ARRAY [1..MAXFORMINGSLAB] OF LREAL;	// Quota Y inizio prima lastra  (CAVALLINA-INCLINATO)
	QuotaZinizioLastra : ARRAY [1..MAXFORMINGSLAB] OF LREAL;	// Quota Z inizio prima lastra  (CAVALLINA-INCLINATO)
	
	QuotaYinizioLastra_A_B : ARRAY [1..MAXFORMINGSLAB] OF ES_SpesoreLastra_A_B;	// Quota Y inizio prima lastra  (CAVALLINA-INCLINATO)
	QuotaZinizioLastra_A_B : ARRAY [1..MAXFORMINGSLAB] OF ES_SpesoreLastra_A_B;	// Quota Z inizio prima lastra  (CAVALLINA-INCLINATO)
	
	numeroLastre_int : UINT;									// Numero lastre per lato cavallina considerando la dimensione L_Utile1 (int)  (CAVALLINA-CASSA)
	
	(* Variabili di supporto *)
	counter1: UINT := 0;	// contatore per ciclo creazione formatura
	counter2: UINT := 0;	// contatore per ciclo creazione formatura
	varEven : UINT := 0;	// Pari o dispari per lato destro (dispari) o lato sinistro (pari) cavallina
	
	(* Variabili di uscita della posizione del punto interno, centrale ed esterno della lastra *)
	XInternoLastra : ARRAY [1..MAXFORMINGSLAB] OF LREAL;		// Coordinata X punto interno n-esima lastra depositata  (CAVALLINA-CASSA)
	YInternoLastra : ARRAY [1..MAXFORMINGSLAB] OF LREAL;		// Coordinata Y punto interno n-esima lastra depositata  (CAVALLINA-CASSA)
	ZInternoLastra : ARRAY [1..MAXFORMINGSLAB] OF LREAL;		// Coordinata Z punto interno n-esima lastra depositata  (CAVALLINA-CASSA)
	XCentroLastra  : ARRAY [1..MAXFORMINGSLAB] OF LREAL;		// Coordinata X punto centrale n-esima lastra depositata  (CAVALLINA-CASSA)
	YCentroLastra  : ARRAY [1..MAXFORMINGSLAB] OF LREAL;		// Coordinata Y punto centrale n-esima lastra depositata  (CAVALLINA-CASSA)
	ZCentroLastra  : ARRAY [1..MAXFORMINGSLAB] OF LREAL;		// Coordinata Z punto centrale n-esima lastra depositata  (CAVALLINA-CASSA)
	XEsternoLastra : ARRAY [1..MAXFORMINGSLAB] OF LREAL;		// Coordinata X punto esterno n-esima lastra depositata  (CAVALLINA-CASSA)
	YEsternoLastra : ARRAY [1..MAXFORMINGSLAB] OF LREAL;		// Coordinata Y punto esterno n-esima lastra depositata  (CAVALLINA-CASSA)
	ZEsternoLastra : ARRAY [1..MAXFORMINGSLAB] OF LREAL;		// Coordinata Z punto esterno n-esima lastra depositata  (CAVALLINA-CASSA)
	
	(* Variabili di uscita della posizione del punto interno, centrale ed esterno della lastra *)
	XInternoLastra_A_B : ARRAY [1..MAXFORMINGSLAB] OF ES_SpesoreLastra_A_B;		// Coordinata X punto interno n-esima lastra depositata  (CAVALLINA-CASSA)
	YInternoLastra_A_B : ARRAY [1..MAXFORMINGSLAB] OF ES_SpesoreLastra_A_B;		// Coordinata Y punto interno n-esima lastra depositata  (CAVALLINA-CASSA)
	ZInternoLastra_A_B : ARRAY [1..MAXFORMINGSLAB] OF ES_SpesoreLastra_A_B;		// Coordinata Z punto interno n-esima lastra depositata  (CAVALLINA-CASSA)
	XCentroLastra_A_B  : ARRAY [1..MAXFORMINGSLAB] OF ES_SpesoreLastra_A_B;		// Coordinata X punto centrale n-esima lastra depositata  (CAVALLINA-CASSA)
	YCentroLastra_A_B  : ARRAY [1..MAXFORMINGSLAB] OF ES_SpesoreLastra_A_B;		// Coordinata Y punto centrale n-esima lastra depositata  (CAVALLINA-CASSA)
	ZCentroLastra_A_B  : ARRAY [1..MAXFORMINGSLAB] OF ES_SpesoreLastra_A_B;		// Coordinata Z punto centrale n-esima lastra depositata  (CAVALLINA-CASSA)
	XEsternoLastra_A_B : ARRAY [1..MAXFORMINGSLAB] OF ES_SpesoreLastra_A_B;		// Coordinata X punto esterno n-esima lastra depositata  (CAVALLINA-CASSA)
	YEsternoLastra_A_B : ARRAY [1..MAXFORMINGSLAB] OF ES_SpesoreLastra_A_B;		// Coordinata Y punto esterno n-esima lastra depositata  (CAVALLINA-CASSA)
	ZEsternoLastra_A_B : ARRAY [1..MAXFORMINGSLAB] OF ES_SpesoreLastra_A_B;		// Coordinata Z punto esterno n-esima lastra depositata  (CAVALLINA-CASSA)

	P_TextModeWrite : P_TextModeWrite;
	MemoriaInizializzata 		:    BOOL;
	NuPiezasLadoDx 				: INT ;
	NuPiezasLadoSx 				: INT ;
	CalForCavallete				: UINT;
	F_ini						: UINT;
	F_Fin						: UINT;
	
	CntLados					: UINT;
	LadoRegistarFor				: UINT;
	NuPieza_A					: UINT;
	NuPieza_B					: UINT;
	LadoA						: UINT;
	LadoB						: UINT;
	
	Fb_CalculoFormaciones 					: Fb_CalculoCoordenadasFinalesFormacion ;
	Fb_CalculoFormacionesTodo0_grados 		: Fb_Fb_CalculoTodo0CoordenadasFinales ;
	Fb_CalculoFormacionesTodo180_grados 	: Fb_CalculoTodo180CoordenadasFinales ;
	Contador: UINT;
	OFSDE_Z180: INT;
	OFSDE_X180: INT;
	OFSDE_Y0: INT;
	OFSDE_Z0: INT;
	OFSDE_J0: INT;
	XDim: INT;
END_VAR

VAR CONSTANT
END_VAR

// Pulisco le variabili interne e le variabili di uscita del FB
IF PulisciMemoria AND NOT PulisciMemoriaDone THEN		// Pulizia delle variabili locali e di uscita
	PulisciMemoriaDone := TRUE;
	memset(ADR(XFinale), 0 , SIZEOF(XFinale));memset(ADR(YFinale), 0 , SIZEOF(YFinale));memset(ADR(ZFinale), 0 , SIZEOF(ZFinale));memset(ADR(JFinale), 0 , SIZEOF(JFinale));
	//###########################################
	memset(ADR(XFinaleLado_0Grados), 0 , SIZEOF(XFinaleLado_0Grados));memset(ADR(YFinaleLado_0Grados), 0 , SIZEOF(YFinaleLado_0Grados));memset(ADR(ZFinaleLado_0Grados), 0 , SIZEOF(ZFinaleLado_0Grados));memset(ADR(JFinaleLado_0Grados), 0 , SIZEOF(JFinaleLado_0Grados));
	memset(ADR(XFinaleLado_180Grados), 0 , SIZEOF(XFinaleLado_180Grados));memset(ADR(YFinaleLado_180Grados), 0 , SIZEOF(YFinaleLado_180Grados));memset(ADR(ZFinaleLado_180Grados), 0 , SIZEOF(ZFinaleLado_180Grados));memset(ADR(JFinaleLado_180Grados), 0 , SIZEOF(JFinaleLado_180Grados));
	memset(ADR(CoorFinaleLado_Pri0_Des180), 0 , SIZEOF(CoorFinaleLado_Pri0_Des180));
	//###########################################################################################
	memset(ADR(FormingSlab), 0 , SIZEOF(FormingSlab));
	memset(ADR(Errore), 0 , SIZEOF(Errore));
	memset(ADR(OrdineDepositoSxDx), 0 , SIZEOF(OrdineDepositoSxDx));
	
	memset(ADR(Spessore_Lastra_Inclinata), 0 , SIZEOF(Spessore_Lastra_Inclinata));memset(ADR(Spessore_Lastra_Inclinata_Cumulato), 0 , SIZEOF(Spessore_Lastra_Inclinata_Cumulato));
	memset(ADR(Spessore_Lastra_Inclinata_lado_A_B), 0 , SIZEOF(Spessore_Lastra_Inclinata_lado_A_B));memset(ADR(Spessore_Lastra_Inclinata_Cumulato_A_B), 0 , SIZEOF(Spessore_Lastra_Inclinata_Cumulato_A_B));
	
	memset(ADR(Spessore_Lastra), 0 , SIZEOF(Spessore_Lastra));memset(ADR(Spessore_Lastra_Cumulato), 0 , SIZEOF(Spessore_Lastra_Cumulato));
	memset(ADR(YCoordinataAppoggioLastra), 0 , SIZEOF(YCoordinataAppoggioLastra));memset(ADR(ZCoordinataAppoggioLastra), 0 , SIZEOF(ZCoordinataAppoggioLastra));
	
	memset(ADR(B), 0 , SIZEOF(B));memset(ADR(b1), 0 , SIZEOF(b1));memset(ADR(h1), 0 , SIZEOF(h1));
	memset(ADR(Yd1), 0 , SIZEOF(Yd1));memset(ADR(Zd1), 0 , SIZEOF(Zd1));
	memset(ADR(Yd2), 0 , SIZEOF(Yd2));memset(ADR(Zd2), 0 , SIZEOF(Zd2));
	memset(ADR(Yd3), 0 , SIZEOF(Yd3));memset(ADR(Zd3), 0 , SIZEOF(Zd3));
	memset(ADR(CI), 0 , SIZEOF(CI));
	memset(ADR(AngoloAlfa_rad), 0 , SIZEOF(AngoloAlfa_rad));memset(ADR(AngoloBeta_rad), 0 , SIZEOF(AngoloBeta_rad));
	
	memset(ADR(QuotaYinizioLastra), 0 , SIZEOF(QuotaYinizioLastra));memset(ADR(QuotaZinizioLastra), 0 , SIZEOF(QuotaZinizioLastra));
	memset(ADR(QuotaYinizioLastra_A_B), 0 , SIZEOF(QuotaYinizioLastra_A_B));memset(ADR(QuotaZinizioLastra_A_B), 0 , SIZEOF(QuotaZinizioLastra_A_B));
	
	memset(ADR(numeroLastre_int), 0 , SIZEOF(numeroLastre_int));
	memset(ADR(XInternoLastra), 0 , SIZEOF(XInternoLastra));memset(ADR(YInternoLastra), 0 , SIZEOF(YInternoLastra));memset(ADR(ZInternoLastra), 0 , SIZEOF(ZInternoLastra));
	memset(ADR(XCentroLastra), 0 , SIZEOF(XCentroLastra));memset(ADR(YCentroLastra), 0 , SIZEOF(YCentroLastra));memset(ADR(ZCentroLastra), 0 , SIZEOF(ZCentroLastra));
	memset(ADR(XEsternoLastra), 0 , SIZEOF(XEsternoLastra));memset(ADR(YEsternoLastra), 0 , SIZEOF(YEsternoLastra));memset(ADR(ZEsternoLastra), 0 , SIZEOF(ZEsternoLastra));
	memset(ADR(Supporto), 0 , SIZEOF(Supporto));
	memset(ADR(Materiale), 0 , SIZEOF(Materiale));
	memset(ADR(TipoElementoDep), 99 , SIZEOF(TipoElementoDep));
	Errore := 0;
	HabiCalTodasCordenadas := FALSE ;
	MemoriaInizializzata := TRUE;
ELSIF NOT PulisciMemoria AND PulisciMemoriaDone THEN
	PulisciMemoriaDone := FALSE;
END_IF

// Calcolo la Formatura, tipo Cassa o Cavallina e salvo su file i risultati ottenuti
IF CalcolaFormatura AND NOT CalcolaFormaturaDone AND MemoriaInizializzata THEN
	// Pulisco le variabili interne e le variabili di uscita del FB
	memset(ADR(XFinale), 0 , SIZEOF(XFinale));memset(ADR(YFinale), 0 , SIZEOF(YFinale));memset(ADR(ZFinale), 0 , SIZEOF(ZFinale));memset(ADR(JFinale), 0 , SIZEOF(JFinale));
	memset(ADR(FormingSlab), 0 , SIZEOF(FormingSlab));
	memset(ADR(Errore), 0 , SIZEOF(Errore));
	memset(ADR(OrdineDepositoSxDx), 0 , SIZEOF(OrdineDepositoSxDx));
	memset(ADR(Spessore_Lastra_Inclinata), 0 , SIZEOF(Spessore_Lastra_Inclinata));memset(ADR(Spessore_Lastra_Inclinata_Cumulato), 0 , SIZEOF(Spessore_Lastra_Inclinata_Cumulato));
	memset(ADR(Spessore_Lastra), 0 , SIZEOF(Spessore_Lastra));memset(ADR(Spessore_Lastra_Cumulato), 0 , SIZEOF(Spessore_Lastra_Cumulato));
	memset(ADR(YCoordinataAppoggioLastra), 0 , SIZEOF(YCoordinataAppoggioLastra));memset(ADR(ZCoordinataAppoggioLastra), 0 , SIZEOF(ZCoordinataAppoggioLastra));
	memset(ADR(B), 0 , SIZEOF(B));memset(ADR(b1), 0 , SIZEOF(b1));memset(ADR(h1), 0 , SIZEOF(h1));
	memset(ADR(Yd1), 0 , SIZEOF(Yd1));memset(ADR(Zd1), 0 , SIZEOF(Zd1));
	memset(ADR(Yd1_A_B), 0 , SIZEOF(Yd1_A_B));memset(ADR(Zd1_A_B), 0 , SIZEOF(Zd1_A_B));
	
	memset(ADR(Yd2), 0 , SIZEOF(Yd2));memset(ADR(Zd2), 0 , SIZEOF(Zd2));
	memset(ADR(Yd2_A_B), 0 , SIZEOF(Yd2_A_B));memset(ADR(Zd2_A_B), 0 , SIZEOF(Zd2_A_B));
	
	memset(ADR(Yd3), 0 , SIZEOF(Yd3));memset(ADR(Zd3), 0 , SIZEOF(Zd3));
	memset(ADR(Yd3_A_B), 0 , SIZEOF(Yd3_A_B));memset(ADR(Zd3_A_B), 0 , SIZEOF(Zd3_A_B));
	
	memset(ADR(CI), 0 , SIZEOF(CI));
	memset(ADR(CI_A_B), 0 , SIZEOF(CI_A_B));
	
	memset(ADR(AngoloAlfa_rad), 0 , SIZEOF(AngoloAlfa_rad));memset(ADR(AngoloBeta_rad), 0 , SIZEOF(AngoloBeta_rad));
	
	memset(ADR(QuotaYinizioLastra), 0 , SIZEOF(QuotaYinizioLastra));memset(ADR(QuotaZinizioLastra), 0 , SIZEOF(QuotaZinizioLastra));
	memset(ADR(QuotaYinizioLastra_A_B), 0 , SIZEOF(QuotaYinizioLastra_A_B));memset(ADR(QuotaZinizioLastra_A_B), 0 , SIZEOF(QuotaZinizioLastra_A_B));
	
	memset(ADR(numeroLastre_int), 0 , SIZEOF(numeroLastre_int));
	
	memset(ADR(XInternoLastra), 0 , SIZEOF(XInternoLastra));memset(ADR(YInternoLastra), 0 , SIZEOF(YInternoLastra));memset(ADR(ZInternoLastra), 0 , SIZEOF(ZInternoLastra));
	memset(ADR(XInternoLastra_A_B), 0 , SIZEOF(XInternoLastra_A_B));memset(ADR(YInternoLastra_A_B), 0 , SIZEOF(YInternoLastra_A_B));memset(ADR(ZInternoLastra_A_B), 0 , SIZEOF(ZInternoLastra_A_B));
	
	memset(ADR(XCentroLastra), 0 , SIZEOF(XCentroLastra));memset(ADR(YCentroLastra), 0 , SIZEOF(YCentroLastra));memset(ADR(ZCentroLastra), 0 , SIZEOF(ZCentroLastra));
	memset(ADR(XCentroLastra_A_B), 0 , SIZEOF(XCentroLastra_A_B));memset(ADR(YCentroLastra_A_B), 0 , SIZEOF(YCentroLastra_A_B));memset(ADR(ZCentroLastra_A_B), 0 , SIZEOF(ZCentroLastra_A_B));
	
	memset(ADR(XEsternoLastra), 0 , SIZEOF(XEsternoLastra));memset(ADR(YEsternoLastra), 0 , SIZEOF(YEsternoLastra));memset(ADR(ZEsternoLastra), 0 , SIZEOF(ZEsternoLastra));
	memset(ADR(XEsternoLastra), 0 , SIZEOF(XEsternoLastra_A_B));memset(ADR(YEsternoLastra_A_B), 0 , SIZEOF(YEsternoLastra_A_B));memset(ADR(ZEsternoLastra_A_B), 0 , SIZEOF(ZEsternoLastra_A_B));

	// Definizione del tipo di deposito a seconda del tipo di supporto utilizzato
	CASE Supporto.Tipologia OF
		PALLET_STANDARD : TipoDeposito := ORIZZONTALE;
		CASSA_STANDARD 	: TipoDeposito := ORIZZONTALE;
		CAVALLETTO 		: TipoDeposito := INCLINATO ; TipoRisultato := TipoLLenarCavellete ;
		BUNDLE 			: TipoDeposito := INCLINATO ; TipoRisultato := TipoLLenarCavellete;//INCLINATO_LATOSINGOLO;
	END_CASE
	
	CASE TipoDeposito OF
		ORIZZONTALE:				// Tipo deposito Orizzontale (Cassa o Pallet)
			(* CASO DELLA CASSA/PALLET CON DEPOSITO ORIZZONTALE *)
			
			(* Creo un ordine di deposito generico, per effettuare i test del singolo lato della cavallina, per debug  *)
			numeroLastre_int := 0;
			FOR counter1:=1 TO MAXFORMINGSLAB BY 1 DO
				IF (TipoElementoDep[counter1] <> e_Tipo_Elemento_Da_Lavorare.NOT_DEFINED AND TipoElementoDep[counter1] <> TERMINATORE) THEN
					numeroLastre_int := numeroLastre_int+1;
				END_IF;
			END_FOR
			
			(* Controlli dati coerenti *)
			IF (Supporto.HMAX <= 0 ) 	OR (Supporto.YDim <= 0 ) THEN
				Errore := ErrValori;
			END_IF
			
			IF (Supporto.ZDim <= 0) THEN
				Errore := ErrHBaseInternaNulla;
				RETURN;
			END_IF
			
			IF (Supporto.XDim <= 0) THEN
				Errore := ErroreLBaseNulla;
				RETURN;
			END_IF
			
			FOR counter1 :=1 TO numeroLastre_int DO
				IF (Supporto.YDim+30 <= Materiale[TipoElementoDep[counter1]].YDim) OR (Supporto.XDim+30 <= Materiale[TipoElementoDep[counter1]].XDim) THEN
					Errore := ErrDimensioneCassa;
				RETURN;
				END_IF
			END_FOR
			
			memset(ADR(Spessore_Lastra), 0 , SIZEOF(Spessore_Lastra));
			FOR counter2 := 1 TO MAXFORMINGSLAB BY 1 DO
				IF CalculoEstacionPickinPiezasDiferentes THEN
					Spessore_Lastra[counter2] := DimensionesPiezasDifEsPiking[counter2].Dim_Horizontal.ZDim;
				ELSE 
					Spessore_Lastra[counter2] := Materiale[TipoElementoDep[counter2]].ZDim;
				END_IF
				
			END_FOR
			
			// Calcola lo spessore complessivo fino al passo n delle lastre/falde depositate sul singolo lato della cavallina 
			memset(ADR(Spessore_Lastra_Cumulato), 0 , SIZEOF(Spessore_Lastra_Cumulato));
			IF (Spessore_Lastra_Cumulato[1] = 0) THEN
				FOR counter2:=1 TO MAXFORMINGSLAB BY 1 DO
					FOR counter1 := 1 TO counter2 BY 1 DO
						Spessore_Lastra_Cumulato[counter2] := Spessore_Lastra_Cumulato[counter2] + Spessore_Lastra[counter1];
					END_FOR
				END_FOR
			END_IF
			
			// Numero di possibili lastre sulla cassa (minore dell'altezza massima)
			FOR counter1:=1 TO MAXFORMINGSLAB BY 1 DO
				IF (TipoElementoDep[counter1] <> e_Tipo_Elemento_Da_Lavorare.NOT_DEFINED AND TipoElementoDep[counter1] <> TERMINATORE) AND ((Spessore_Lastra_Cumulato[counter1] >0) AND 
					(Spessore_Lastra_Cumulato[counter1]+Supporto.ZDim < Supporto.HMAX)) THEN
						numeroLastre_int := counter1;
				END_IF
				IF (Spessore_Lastra_Cumulato[counter1]+Supporto.ZDim >= Supporto.HMAX) AND Supporto.Tipologia <> PALLET_STANDARD AND counter1 <= numeroLastre_int THEN
					Errore := ErrNumeroPezzi;
				END_IF
			END_FOR
			
			// Calcolo il punto Z interno, centrale ed esterno per ogni lastra posizionata sulla cassa
			FOR counter1:=1 TO numeroLastre_int BY 1 DO
				ZInternoLastra[counter1] := Supporto.ZDim + Spessore_Lastra_Cumulato[counter1-1];
				ZCentroLastra[counter1] := Supporto.ZDim + (Spessore_Lastra_Cumulato[counter1-1] + Spessore_Lastra_Cumulato[counter1]) / 2;
				ZEsternoLastra[counter1] := Supporto.ZDim + Spessore_Lastra_Cumulato[counter1];
			END_FOR
			
			(* Pulisco le uscite e setto a TERMINATORE tutti gli elementi di FormingSlab *)
			memset(ADR(XFinale),0,SIZEOF(XFinale));memset(ADR(YFinale),0,SIZEOF(YFinale));memset(ADR(ZFinale),0,SIZEOF(ZFinale));memset(ADR(JFinale),0,SIZEOF(JFinale));
			memset(ADR(FormingSlab),0,SIZEOF(FormingSlab));
			FOR counter1 := 1 TO MAXFORMINGSLAB DO
				FormingSlab.PElement[counter1].Typology := TERMINATORE;
			END_FOR
			
			(* Calcolo delle coordinate X,Y,Z del punto finale sulla base del TipoRisultato *)
			FOR counter2:=1 TO numeroLastre_int BY 1 DO
				XInternoLastra[counter2] := 0; YInternoLastra[counter2] := 0;
				XCentroLastra[counter2] := 0;  YCentroLastra[counter2] := 0;
				XEsternoLastra[counter2] := 0; YEsternoLastra[counter2] := 0;
				
				CASE TipoRisultato OF
					1:	XFinale[counter2] := XInternoLastra[counter2] + Supporto.OFSDE_X90;
						YFinale[counter2] := YInternoLastra[counter2] + Supporto.OFSDE_Y90;
						ZFinale[counter2] := ZInternoLastra[counter2] + Supporto.OFSDE_Z90;
						JFinale[counter2] := 90 + Supporto.OFSDE_J90;
					2:	XFinale[counter2] := XCentroLastra[counter2] + Supporto.OFSDE_X90;
						YFinale[counter2] := YCentroLastra[counter2] + Supporto.OFSDE_Y90;
						ZFinale[counter2] := ZCentroLastra[counter2] + Supporto.OFSDE_Z90;
						JFinale[counter2] := 90  + Supporto.OFSDE_J90;
					3:	XFinale[counter2] := XEsternoLastra[counter2] + Supporto.OFSDE_X90;
						YFinale[counter2] := YEsternoLastra[counter2] + Supporto.OFSDE_Y90;
						ZFinale[counter2] := ZEsternoLastra[counter2] + Supporto.OFSDE_Z90;
						JFinale[counter2] := 90 + Supporto.OFSDE_J90;	
				END_CASE
				
			END_FOR;
			FOR counter1:=1 TO numeroLastre_int BY 1 DO
				FormingSlab.Enable := 1;										// Abilitato
				//FormingSlab.Code[1] := 1;
				//FormingSlab.PElement[counter1].Typology := Materiale[OrdineDeposito[counter1]].Typology;

				//Indico la tipologia di elemnto che vado a depositare in base all'ordine passato dall'esterno
				CASE TipoElementoDep[counter1] OF
					LASTRA:
						FormingSlab.PElement[counter1].Typology := LASTRA;

					FALDA:
						FormingSlab.PElement[counter1].Typology := FALDA;

					TERMINATORE:
						FormingSlab.PElement[counter1].Typology := TERMINATORE;
				
				ELSE
					FormingSlab.PElement[counter1].Typology := e_Tipo_Elemento_Da_Lavorare.NOT_DEFINED;

				END_CASE
				IF CalculoEstacionPickinPiezasDiferentes THEN 
					FormingSlab.PElement[counter1].XDim := DimensionesPiezasDifEsPiking[counter1].Dim_Horizontal.XDim;		// Dimensione X Lastra		
					FormingSlab.PElement[counter1].YDim := DimensionesPiezasDifEsPiking[counter1].Dim_Horizontal.YDim;		// Dimensione Y Lastra
					FormingSlab.PElement[counter1].ZDim := DimensionesPiezasDifEsPiking[counter1].Dim_Horizontal.ZDim;		// Dimensione Z Lastra
				ELSE
					FormingSlab.PElement[counter1].XDim := Materiale[TipoElementoDep[counter1]].XDim;		// Dimensione X Lastra		
					FormingSlab.PElement[counter1].YDim := Materiale[TipoElementoDep[counter1]].YDim;		// Dimensione Y Lastra
					FormingSlab.PElement[counter1].ZDim := Materiale[TipoElementoDep[counter1]].ZDim;		// Dimensione Z Lastra
				END_IF
				FormingSlab.PElement[counter1].X := XFinale[counter1];
				FormingSlab.PElement[counter1].Y := YFinale[counter1];
				FormingSlab.PElement[counter1].Z := ZFinale[counter1];
				FormingSlab.PElement[counter1].J := JFinale[counter1];
			END_FOR
		
			
		
		INCLINATO:					// Tipo deposito inclinato ( Cavallina)
			(* CASO DELLA CAVALLINA CON DEPOSITO INCLINATO DAI DUE LATI*)
			
			numeroLastre_int := 0;
			FOR counter1:=1 TO MAXFORMINGSLAB/2 BY 1 DO
				IF (TipoElementoDep[counter1] <> e_Tipo_Elemento_Da_Lavorare.NOT_DEFINED AND TipoElementoDep[counter1] <> TERMINATORE) THEN
					numeroLastre_int := numeroLastre_int+1;
				END_IF;
			END_FOR
	
			(* Replico l'ordine di deposito del singolo lato su entrambi i lati, sx e dx della cavallina *)
			FOR counter1:=1 TO MAXFORMINGSLAB BY 1 DO
				varEven := counter1 MOD 2;
				CASE varEven OF
					0:	
						OrdineDepositoSxDx[counter1] := TipoElementoDep[counter1];//OrdineDeposito[counter1/2];
					1:	
						OrdineDepositoSxDx[counter1] := TipoElementoDep[counter1];//OrdineDeposito[(counter1+varEven)/2];
				END_CASE;
			END_FOR;
			
			(* Controlli dati coerenti *)
			FOR counter1:=1 TO MAXFORMINGSLAB DO
				IF(Materiale[TipoElementoDep[counter1]].XDim <0) OR (Materiale[TipoElementoDep[counter1]].YDim <0) OR 
					(Materiale[TipoElementoDep[counter1]].ZDim <0)  OR (Materiale[TipoElementoDep[counter1]].Typology <0) THEN
						Errore := Errvalori;
						RETURN;
				END_IF
			END_FOR
					
			IF Supporto.ZDim <= 0 THEN//OR (Supporto.ZDim_Int2 <=0) THEN
				Errore := ErrHBaseInternaNulla;
				RETURN;
			END_IF
			
			IF Supporto.ZDim_Ext1 <= 0 AND Supporto.TipoPianoAppoggio = 1 THEN//OR (Supporto.ZDim_Ext2 <=0) THEN
				Errore := ErrHBaseEsternaNulla;
				RETURN;
			END_IF
			
			IF Supporto.ZDim > Supporto.ZDim_Ext1 AND Supporto.TipoPianoAppoggio = 1 THEN//OR (Supporto.ZDim_Int2 > Supporto.ZDim_Ext2) THEN
				Errore := ErrBaseInclinata;
				RETURN;
			END_IF
			
			IF (Supporto.HMAX <= 0) THEN		// altezza cavallina
				Errore := ErrHTotaleNulla;
				RETURN;
			END_IF
			
			IF (Supporto.YDim <= 0) THEN		// larghezza Y cavallina
				Errore := ErroreLBaseNulla;
				RETURN;
			END_IF
			
			// Base centrale non utilizzata della cavallina
			IF Supporto.Tipologia = CAVALLETTO    THEN
				B := Supporto.YDim - Supporto.DimBaseUtile - Supporto.DimBaseUtile;
				B2 := ( Supporto.YDim / 2 )-supporto.DimBaseUtile ;
				CorYIz := supporto.DimBaseUtile ;
				CorYDe := Supporto.YDim - supporto.DimBaseUtile ;
				BaseAlgulo := ( Supporto.YDim /2) - (Supporto.DimVertice /2)- supporto.DimBaseUtile;
			ELSE
				B := Supporto.YDim - Supporto.DimBaseUtile - Supporto.DimBaseUtile;
				B2 := ( Supporto.YDim / 2 )-supporto.DimBaseUtile ;
			END_IF
			
			//B := Supporto.YDim - Supporto.DimBaseUtile - Supporto.DimBaseUtile;
			//B2 := ( Supporto.YDim / 2 )-supporto.DimBaseUtile ;
			IF (B <= 0 ) THEN
				Errore := ErrBase;
				RETURN;
			END_IF
			
			IF (Supporto.DimBaseUtile <= 0 ) OR (Supporto.DimBaseUtile <= 0 ) THEN
				Errore := ErrLUtile;
			END_IF
			
			b1 := (B - Supporto.DimVertice) / 2;	// base del triangolo rettangolo dell'angolo alfa
			IF (b1 <= 0 ) THEN
				Errore := ErrBaseAlfa;
				RETURN;
			END_IF
			
			h1 := Supporto.HMAX - Supporto.ZDim; // Altezza del triangolo rettangolo dell'angolo alfa
			IF h1 <= 0 THEN
				Errore := ErrAltezzaAlfa;
				RETURN;
			END_IF
			
			(* calcolo angolo alfa dell'inclinazione appoggio della lastra *)
			AngoloAlfa_rad := ATAN( b1 / h1); // Angolo superiore appoggio cavallina (in radianti)
			AlgoloAlfa_gradi := rad_to_deg(AngoloAlfa_rad); 
			
			IF (AlgoloAlfa_gradi >= 90) THEN
				Errore := ErrAngolo;
				RETURN;
			END_IF
			
			(* Calcolo angolo beta dell'eventuale piano di appoggio inclinato della cavallina*)
			AngoloBeta_rad := ATAN( (Supporto.ZDim_Ext1 - Supporto.ZDim) / Supporto.DimBaseUtile); 	// Angolo del piano di appoggio inclinato della cavallina (in radianti)
			AngoloBeta_gradi := rad_to_deg(AngoloBeta_rad);					// Angolo del piano di appoggio inclinato della cavallina (in gradi)
			rad90 := deg_to_rad(90);
			
			IF (AlgoloAlfa_gradi < (AngoloBeta_gradi-1)) AND FALSE (*Quitar alarma pendiente base*) THEN
				Errore := ErrPendenzaBase;					// Angolo alfa deve essere maggiore dell'angolo beta
				RETURN;
			END_IF
			
			// Calcolo lo spessore di ogni singola lastra/falda depositata sul lato della cavallina
			Spessore_Lastra_Inclinata[1] := 0;
			FOR counter2:=2 TO MAXFORMINGSLAB/2 BY 1 DO
				IF CalculoEstacionPickinPiezasDiferentes AND Supporto.Tipologia = CAVALLETTO THEN 
					Fun_PiezaLadoCaballete(Nu_PiezaGlobal:= counter2 , Grados:= ADR(LadoRegistarFor) , 
														Nu_pieza_LadoA=>NuPieza_A , Nu_pieza_LadoB=> NuPieza_B  );
				CASE Supporto.TipoTrabajoLado_Cavallete OF
					0:
						CASE LadoRegistarFor OF
							0 :
								Spessore_Lastra_Inclinata_lado_A_B[NuPieza_A].Lado_A_0Grados := 
										DimensionesPiezasDifEsPiking[NuPieza_A].DimPieza_LadoA.ZDim / COS(AngoloAlfa_rad);	
						  180 :
								Spessore_Lastra_Inclinata_lado_A_B[NuPieza_B].Lado_B_180Grados := 
										DimensionesPiezasDifEsPiking[NuPieza_B].DimPieza_LadoB.ZDim / COS(AngoloAlfa_rad);
						END_CASE
					1: 
						Spessore_Lastra_Inclinata_lado_A_B[counter2].Lado_A_0Grados := 
										DimensionesPiezasDifEsPiking[counter2-1].DimPieza_LadoA.ZDim / COS(AngoloAlfa_rad);
						;
					2: 
						Spessore_Lastra_Inclinata_lado_A_B[counter2].Lado_B_180Grados := 
										DimensionesPiezasDifEsPiking[counter2-1].DimPieza_LadoB.ZDim / COS(AngoloAlfa_rad);
						;
				END_CASE
				ELSIF	CalculoEstacionPickinPiezasDiferentes  AND Supporto.Tipologia <> CAVALLETTO THEN 
					 Spessore_Lastra_Inclinata[counter2] := DimensionesPiezasDifEsPiking[counter2-1].Dim_Horizontal.ZDim / COS(AngoloAlfa_rad);
				ELSE
					 
					Spessore_Lastra_Inclinata[counter2] := Materiale[TipoElementoDep[counter2-1]].ZDim / COS(AngoloAlfa_rad);
				END_IF
			END_FOR;
			
			// Calcola lo spessore complessivo fino al passo n delle lastre/falde depositate sul singolo lato della cavallina 
			//memset(ADR(Spessore_Lastra_Inclinata_Cumulato), 0 , SIZEOF(Spessore_Lastra_Inclinata_Cumulato));
			IF NOT CalculoEstacionPickinPiezasDiferentes THEN 
				IF (Spessore_Lastra_Inclinata_Cumulato[2] = 0) THEN
					FOR counter2:=1 TO MAXFORMINGSLAB/2 BY 1 DO
						FOR counter1 := 1 TO counter2 BY 1 DO
							Spessore_Lastra_Inclinata_Cumulato[counter2] := Spessore_Lastra_Inclinata_Cumulato[counter2]+Spessore_Lastra_Inclinata[counter1];
						END_FOR
					END_FOR
				END_IF
			END_IF
			IF CalculoEstacionPickinPiezasDiferentes AND Supporto.Tipologia = CAVALLETTO THEN 
				IF (Spessore_Lastra_Inclinata_Cumulato_A_B[2].Lado_A_0Grados = 0) THEN
					FOR counter2:=1 TO MAXFORMINGSLAB/2 BY 1 DO
						FOR counter1 := 1 TO counter2 BY 1 DO
							Spessore_Lastra_Inclinata_Cumulato_A_B[counter2].Lado_A_0Grados := 
												Spessore_Lastra_Inclinata_Cumulato_A_B[counter2].Lado_A_0Grados
														+	Spessore_Lastra_Inclinata_lado_A_B[counter1].Lado_A_0Grados;
							Spessore_Lastra_Inclinata_Cumulato_A_B[counter2].Lado_B_180Grados := 
												Spessore_Lastra_Inclinata_Cumulato_A_B[counter2].Lado_B_180Grados
														+	Spessore_Lastra_Inclinata_lado_A_B[counter1].Lado_B_180Grados;
						END_FOR
					END_FOR
				END_IF
				
			ELSIF CalculoEstacionPickinPiezasDiferentes AND Supporto.Tipologia <> CAVALLETTO THEN 
				Spessore_Lastra_Inclinata_Cumulato[counter2] := 
												Spessore_Lastra_Inclinata_Cumulato[counter2]
														+	Spessore_Lastra_Inclinata[counter1];
			END_IF
			// Numero di possibili lastre sul singolo lato
			//FOR counter1:=1 TO MAXFORMINGSLAB/2 BY 1 DO
				//IF (OrdineDeposito[counter1] <> e_Tipo_Elemento_Da_Lavorare.NOT_DEFINED AND OrdineDeposito[counter1] <> TERMINATORE) AND 
				//	((Spessore_Lastra_Inclinata_Cumulato[counter1] >0) AND (Spessore_Lastra_Inclinata_Cumulato[counter1] < Supporto.DimBaseUtile)) THEN
				//		numeroLastre_int := counter1;
				//END_IF
				//IF (OrdineDeposito[counter1] <> e_Tipo_Elemento_Da_Lavorare.NOT_DEFINED AND OrdineDeposito[counter1] <> TERMINATORE) AND 
				//	(Spessore_Lastra_Inclinata_Cumulato[counter1] >= Supporto.DimBaseUtile) THEN
				//		Errore := ErrNumeroPezzi;	// il supervisore mi ha passato troppe lastre rispetto allo spazio utile
				//END_IF
			//END_FOR
			Fun_NumeroPiezasLadoCaballete(NuPieasTotales:= numeroLastre_int , PiezasLadoA:=ADR(LadoA) , PiezasLadoB:=ADR(LadoB) );
			
			
			IF (Spessore_Lastra_Inclinata_Cumulato[numeroLastre_int] >= Supporto.DimBaseUtile*2) AND NOT CalculoEstacionPickinPiezasDiferentes  THEN
				Errore := ErrNumeroPezzi;	// il supervisore mi ha passato troppe lastre rispetto allo spazio utile
				
				
			ELSIF (Spessore_Lastra_Inclinata_Cumulato_A_B[LadoA].Lado_A_0Grados >= Supporto.DimBaseUtile ) AND  
															CalculoEstacionPickinPiezasDiferentes   THEN 
				Errore := ErrNumeroPezzi;	// il supervisore mi ha passato troppe lastre rispetto allo spazio utile
			ELSIF (Spessore_Lastra_Inclinata_Cumulato_A_B[LadoA].Lado_B_180Grados >= Supporto.DimBaseUtile ) AND  CalculoEstacionPickinPiezasDiferentes   THEN 
				Errore := ErrNumeroPezzi;	// il supervisore mi ha passato troppe lastre rispetto allo spazio utile	
			END_IF
			
			
			
			IF  NOT CalculoEstacionPickinPiezasDiferentes THEN
			// Calcolo lo spostamento del punto centrale e del punto esterno della singola lastra/falda rispetto al punto interno(iniziale) della medesima lastra/falda
				FOR counter2:=1 TO numeroLastre_int BY 1 DO
					Yd1[counter2] := Materiale[TipoElementoDep[counter2]].ZDim / 2 * COS (AngoloAlfa_rad);		// Spostamento Centro lastra da interno lastra in Y
					Zd1[counter2] := Materiale[TipoElementoDep[counter2]].ZDim / 2 * SIN (AngoloAlfa_rad);		// Spostamento Centro lastra da interno lastra in Z
					Yd2[counter2] := Materiale[TipoElementoDep[counter2]].ZDim  * COS (AngoloAlfa_rad);			// Spostamento esterno lastra da interno lastra in Y
					Zd2[counter2] := Materiale[TipoElementoDep[counter2]].ZDim  * SIN (AngoloAlfa_rad);			// Spostamento esterno lastra da interno lastra in Z
				END_FOR
			END_IF
			IF CalculoEstacionPickinPiezasDiferentes THEN
				FOR counter2:=1 TO numeroLastre_int BY 1 DO
					IF Supporto.Tipologia = CAVALLETTO THEN 
						Fun_PiezaLadoCaballete(Nu_PiezaGlobal:=counter2 , Grados:= ADR(LadoRegistarFor)  ,
										 Nu_pieza_LadoA=>NuPieza_A , Nu_pieza_LadoB=> NuPieza_B  );
						CASE Supporto.TipoTrabajoLado_Cavallete  OF
							
							0:
								CASE LadoRegistarFor OF
									0: 
										Yd1_A_B[NuPieza_A].Lado_A_0Grados := DimensionesPiezasDifEsPiking[NuPieza_A].DimPieza_LadoA.ZDim / 2 * COS (AngoloAlfa_rad);		// Spostamento Centro lastra da interno lastra in Y
										Zd1_A_B[NuPieza_A].Lado_A_0Grados := DimensionesPiezasDifEsPiking[NuPieza_A].DimPieza_LadoA.ZDim / 2 * SIN (AngoloAlfa_rad);		// Spostamento Centro lastra da interno lastra in Z
										Yd2_A_B[NuPieza_A].Lado_A_0Grados := DimensionesPiezasDifEsPiking[NuPieza_A].DimPieza_LadoA.ZDim  * COS (AngoloAlfa_rad);			// Spostamento esterno lastra da interno lastra in Y
										Zd1_A_B[NuPieza_A].Lado_A_0Grados := DimensionesPiezasDifEsPiking[NuPieza_A].DimPieza_LadoA.ZDim  * SIN (AngoloAlfa_rad);			// Spostamento esterno lastra da interno lastra in Z
										
								 180: 
										Yd1_A_B[NuPieza_B].Lado_B_180Grados := DimensionesPiezasDifEsPiking[NuPieza_B].DimPieza_LadoB.ZDim / 2 * COS (AngoloAlfa_rad);		// Spostamento Centro lastra da interno lastra in Y
										Zd1_A_B[NuPieza_B].Lado_B_180Grados := DimensionesPiezasDifEsPiking[NuPieza_B].DimPieza_LadoB.ZDim  / 2 * SIN (AngoloAlfa_rad);		// Spostamento Centro lastra da interno lastra in Z
										Yd2_A_B[NuPieza_B].Lado_B_180Grados := DimensionesPiezasDifEsPiking[NuPieza_B].DimPieza_LadoB.ZDim   * COS (AngoloAlfa_rad);			// Spostamento esterno lastra da interno lastra in Y
										Zd1_A_B[NuPieza_B].Lado_B_180Grados := DimensionesPiezasDifEsPiking[NuPieza_B].DimPieza_LadoB.ZDim  * SIN (AngoloAlfa_rad);			// Spostamento esterno lastra da interno lastra in Z	
								END_CASE
							1:
								Yd1_A_B[counter2].Lado_A_0Grados := DimensionesPiezasDifEsPiking[counter2].DimPieza_LadoA.ZDim / 2 * COS (AngoloAlfa_rad);		// Spostamento Centro lastra da interno lastra in Y
								Zd1_A_B[counter2].Lado_A_0Grados := DimensionesPiezasDifEsPiking[counter2].DimPieza_LadoA.ZDim / 2 * SIN (AngoloAlfa_rad);		// Spostamento Centro lastra da interno lastra in Z
								Yd2_A_B[counter2].Lado_A_0Grados := DimensionesPiezasDifEsPiking[counter2].DimPieza_LadoA.ZDim  * COS (AngoloAlfa_rad);			// Spostamento esterno lastra da interno lastra in Y
								Zd1_A_B[counter2].Lado_A_0Grados := DimensionesPiezasDifEsPiking[counter2].DimPieza_LadoA.ZDim  * SIN (AngoloAlfa_rad);			// Spostamento esterno lastra da interno lastra in Z
							
							
							
							2:
								Yd1_A_B[counter2].Lado_B_180Grados := DimensionesPiezasDifEsPiking[counter2].DimPieza_LadoB.ZDim / 2 * COS (AngoloAlfa_rad);		// Spostamento Centro lastra da interno lastra in Y
								Zd1_A_B[counter2].Lado_B_180Grados := DimensionesPiezasDifEsPiking[counter2].DimPieza_LadoB.ZDim  / 2 * SIN (AngoloAlfa_rad);		// Spostamento Centro lastra da interno lastra in Z
								Yd2_A_B[counter2].Lado_B_180Grados := DimensionesPiezasDifEsPiking[counter2].DimPieza_LadoB.ZDim   * COS (AngoloAlfa_rad);			// Spostamento esterno lastra da interno lastra in Y
								Zd1_A_B[counter2].Lado_B_180Grados := DimensionesPiezasDifEsPiking[counter2].DimPieza_LadoB.ZDim  * SIN (AngoloAlfa_rad);			// Spostamento esterno lastra da interno lastra in Z	
						END_CASE
					ELSIF Supporto.Tipologia <> CAVALLETTO THEN 
						Yd1[counter2] := DimensionesPiezasDifEsPiking[counter2].Dim_Horizontal.ZDim/ 2 * COS (AngoloAlfa_rad);		// Spostamento Centro lastra da interno lastra in Y
						Zd1[counter2] := DimensionesPiezasDifEsPiking[counter2].Dim_Horizontal.ZDim/ 2 * SIN (AngoloAlfa_rad);		// Spostamento Centro lastra da interno lastra in Z
						Yd2[counter2] := DimensionesPiezasDifEsPiking[counter2].Dim_Horizontal.ZDim  * COS (AngoloAlfa_rad);			// Spostamento esterno lastra da interno lastra in Y
						Zd1[counter2] := DimensionesPiezasDifEsPiking[counter2].Dim_Horizontal.ZDim  * SIN (AngoloAlfa_rad);			// Spostamento esterno lastra da interno lastra in Z
					END_IF 
				END_FOR
			END_IF
			
			// Calcolo la proiezione mancante di ogni singola lastra/falda; Tramite CI posso calcolare lo spostamento Yd3,Zd3 dovuto al piano inclinato
			// dovuto all'angolo beta. Utilizzo il teorema dei seni per calcolare ogni CI da SLIC
			IF NOT CalculoEstacionPickinPiezasDiferentes THEN
				FOR counter1:=1 TO numeroLastre_int BY 1 DO
					CI[counter1] := (Spessore_Lastra_Inclinata_Cumulato[counter1] * SIN (AngoloBeta_rad) ) / SIN( rad90 + AngoloAlfa_rad - AngoloBeta_rad);
					Yd3[counter1] := -CI[counter1] * SIN(AngoloAlfa_rad);
					Zd3[counter1] := CI[counter1] * COS(AngoloAlfa_rad);
				END_FOR;
			END_IF
			
			IF CalculoEstacionPickinPiezasDiferentes THEN
				FOR counter1:=1 TO numeroLastre_int BY 1 DO
					IF Supporto.Tipologia = CAVALLETTO THEN 
						Fun_PiezaLadoCaballete(Nu_PiezaGlobal:=counter1 , Grados:= ADR(LadoRegistarFor)  ,
										 Nu_pieza_LadoA=>NuPieza_A , Nu_pieza_LadoB=> NuPieza_B  );
						CASE Supporto.TipoTrabajoLado_Cavallete  OF
							0:
								CASE LadoRegistarFor OF
									0: 
										CI_A_B[NuPieza_A].Lado_A_0Grados := (Spessore_Lastra_Inclinata_Cumulato_A_B[NuPieza_A].Lado_A_0Grados * SIN (AngoloBeta_rad) ) / SIN( rad90 + AngoloAlfa_rad - AngoloBeta_rad);
										Yd3_A_B[NuPieza_A].Lado_A_0Grados := -CI[NuPieza_A] * SIN(AngoloAlfa_rad);
										Zd3_A_B[NuPieza_A].Lado_A_0Grados :=  CI[NuPieza_A] * COS(AngoloAlfa_rad);
								 180: 
										CI_A_B[NuPieza_B].Lado_B_180Grados := (Spessore_Lastra_Inclinata_Cumulato_A_B[NuPieza_B].Lado_B_180Grados * SIN (AngoloBeta_rad) ) / SIN( rad90 + AngoloAlfa_rad - AngoloBeta_rad);
										Yd3_A_B[NuPieza_B].Lado_B_180Grados := -CI[NuPieza_B] * SIN(AngoloAlfa_rad);
										Zd3_A_B[NuPieza_B].Lado_B_180Grados :=  CI[NuPieza_B] * COS(AngoloAlfa_rad);
								END_CASE
							1:
								CI_A_B[counter1].Lado_A_0Grados := (Spessore_Lastra_Inclinata_Cumulato_A_B[counter1].Lado_A_0Grados * SIN (AngoloBeta_rad) ) / SIN( rad90 + AngoloAlfa_rad - AngoloBeta_rad);
								Yd3_A_B[counter1].Lado_A_0Grados := -CI[counter1] * SIN(AngoloAlfa_rad);
								Zd3_A_B[counter1].Lado_A_0Grados :=  CI[counter1] * COS(AngoloAlfa_rad);
							2:
								CI_A_B[counter1].Lado_B_180Grados := (Spessore_Lastra_Inclinata_Cumulato_A_B[NuPieza_B].Lado_B_180Grados * SIN (AngoloBeta_rad) ) / SIN( rad90 + AngoloAlfa_rad - AngoloBeta_rad);
								Yd3_A_B[counter1].Lado_B_180Grados := -CI[counter1] * SIN(AngoloAlfa_rad);
								Zd3_A_B[counter1].Lado_B_180Grados :=  CI[counter1] * COS(AngoloAlfa_rad);
						END_CASE
					ELSIF Supporto.Tipologia <> CAVALLETTO THEN 
						CI[counter1] := (Spessore_Lastra_Inclinata_Cumulato[counter1] * SIN (AngoloBeta_rad) ) / SIN( rad90 + AngoloAlfa_rad - AngoloBeta_rad);
						Yd3[counter1] := -CI[counter1] * SIN(AngoloAlfa_rad);
						Zd3[counter1] := CI[counter1] * COS(AngoloAlfa_rad);
					END_IF
				END_FOR;
			END_IF
			// Quota Y e Z del punto di appoggio di ogni lastra sulla cavallina
			// Quota Y e Z del punto interno centrale di ogni lastra; corrisponde a YInternoLastra e ZInternoLastra
			IF NOT CalculoEstacionPickinPiezasDiferentes THEN
				NuPiezasLadoDx := 0 ;
				NuPiezasLadoSx := 0 ;
				FOR counter2:=1 TO numeroLastre_int BY 1 DO
					XInternoLastra[counter2] := Supporto.XDim/2;
					varEven := counter2 MOD 2;
					IF Supporto.Tipologia = CAVALLETTO    THEN
						CASE varEven OF
							0:	
									CASE TipoCalculo OF
									0:
										YCoordinataAppoggioLastra[counter2] := (B/2) + Spessore_Lastra_Inclinata_Cumulato[counter2] + Yd3[counter2];
										
									
									1: 
										NuPiezasLadoDx := NuPiezasLadoDx +1 ;
										YCoordinataAppoggioLastra[counter2] := (CorYDe) + Spessore_Lastra_Inclinata_Cumulato[NuPiezasLadoDx] + Yd3[NuPiezasLadoDx];
										
									END_CASE
							1:
								CASE TipoCalculo OF
									0:
										YCoordinataAppoggioLastra[counter2] := (B/2) + Spessore_Lastra_Inclinata_Cumulato[counter2] - Yd3[counter2];
									
									1:
										NuPiezasLadoSx := NuPiezasLadoSx + 1;
										YCoordinataAppoggioLastra[counter2] := (CorYIz) + Spessore_Lastra_Inclinata_Cumulato[NuPiezasLadoSx] - Yd3[NuPiezasLadoSx];
								END_CASE
						END_CASE
						
						
						ELSE
						YCoordinataAppoggioLastra[counter2] := (B/2) + Spessore_Lastra_Inclinata_Cumulato[counter2] + Yd3[counter2];
							
					END_IF
					//YCoordinataAppoggioLastra[counter2] := (*(B2) +*) Spessore_Lastra_Inclinata_Cumulato[counter2] + Yd3[counter2];
					YInternoLastra[counter2] := YCoordinataAppoggioLastra[counter2] - (Materiale[TipoElementoDep[counter2]].YDim / 2) * SIN (AngoloAlfa_rad);
					ZCoordinataAppoggioLastra[counter2] := Supporto.ZDim + Zd3[counter2];
					ZInternoLastra[counter2] := ZCoordinataAppoggioLastra[counter2] + (Materiale[TipoElementoDep[counter2]].YDim / 2) * COS (AngoloAlfa_rad); 
				END_FOR
			END_IF
			IF CalculoEstacionPickinPiezasDiferentes THEN
				FOR counter2:=1 TO numeroLastre_int BY 1 DO
					XInternoLastra[counter2] := Supporto.XDim/2;
					Fun_PiezaLadoCaballete(Nu_PiezaGlobal:= counter2 , Grados:= ADR(LadoRegistarFor)  ,
										 Nu_pieza_LadoA=>NuPieza_A , Nu_pieza_LadoB=> NuPieza_B  );
					IF Supporto.Tipologia = CAVALLETTO    THEN
						CASE Supporto.TipoTrabajoLado_Cavallete  OF
							0:	
								CASE LadoRegistarFor OF
									0: 
										YCoordinataAppoggioLastra_A_B[NuPieza_A].Lado_A_0Grados := (B/2) + Spessore_Lastra_Inclinata_Cumulato_A_B[NuPieza_A].Lado_A_0Grados + Yd3[NuPieza_A];
										YInternoLastra_A_B[NuPieza_A].Lado_A_0Grados := YCoordinataAppoggioLastra_A_B[NuPieza_A].Lado_A_0Grados - (DimensionesPiezasDifEsPiking[NuPieza_A].DimPieza_LadoA.YDim / 2) * SIN (AngoloAlfa_rad);
										ZCoordinataAppoggioLastra_A_B[NuPieza_A].Lado_A_0Grados := Supporto.ZDim + Zd3_A_B[NuPieza_A].Lado_A_0Grados;
										ZInternoLastra_A_B[counter2].Lado_A_0Grados := ZCoordinataAppoggioLastra_A_B[counter2].Lado_A_0Grados + (DimensionesPiezasDifEsPiking[counter2].Dim_Horizontal.YDim / 2) * COS (AngoloAlfa_rad); 	
									180:
										YCoordinataAppoggioLastra_A_B[NuPieza_B].Lado_B_180Grados := (B/2) + Spessore_Lastra_Inclinata_Cumulato_A_B[NuPieza_B].Lado_B_180Grados + Yd3[NuPieza_B];
										YInternoLastra_A_B[NuPieza_B].Lado_B_180Grados := YCoordinataAppoggioLastra_A_B[NuPieza_B].Lado_B_180Grados - (DimensionesPiezasDifEsPiking[NuPieza_B].DimPieza_LadoB.YDim / 2) * SIN (AngoloAlfa_rad);
										ZCoordinataAppoggioLastra_A_B[NuPieza_B].Lado_B_180Grados := Supporto.ZDim + Zd3_A_B[NuPieza_B].Lado_B_180Grados;
										ZInternoLastra_A_B[NuPieza_B].Lado_B_180Grados := ZCoordinataAppoggioLastra_A_B[NuPieza_B].Lado_B_180Grados + (DimensionesPiezasDifEsPiking[NuPieza_A].DimPieza_LadoB.YDim / 2) * COS (AngoloAlfa_rad); 	
								END_CASE
							1: 
								YCoordinataAppoggioLastra_A_B[counter2].Lado_A_0Grados := (B/2) + Spessore_Lastra_Inclinata_Cumulato_A_B[counter2].Lado_B_180Grados + Yd3[counter2];
								YInternoLastra_A_B[counter2].Lado_A_0Grados := YCoordinataAppoggioLastra_A_B[counter2].Lado_A_0Grados - (DimensionesPiezasDifEsPiking[counter2].DimPieza_LadoA.YDim / 2) * SIN (AngoloAlfa_rad);
								ZCoordinataAppoggioLastra_A_B[counter2].Lado_A_0Grados := Supporto.ZDim + Zd3_A_B[counter2].Lado_A_0Grados;
								ZInternoLastra_A_B[counter2].Lado_A_0Grados := ZCoordinataAppoggioLastra_A_B[counter2].Lado_A_0Grados + (DimensionesPiezasDifEsPiking[counter2].Dim_Horizontal.YDim / 2) * COS (AngoloAlfa_rad); 
							2:
								YCoordinataAppoggioLastra_A_B[counter2].Lado_B_180Grados := (B/2) + Spessore_Lastra_Inclinata_Cumulato_A_B[counter2].Lado_B_180Grados + Yd3[NuPieza_B];
								YInternoLastra_A_B[counter2].Lado_B_180Grados := YCoordinataAppoggioLastra_A_B[counter2].Lado_B_180Grados - (DimensionesPiezasDifEsPiking[counter2].DimPieza_LadoB.YDim / 2) * SIN (AngoloAlfa_rad);
								ZCoordinataAppoggioLastra_A_B[counter2].Lado_B_180Grados := Supporto.ZDim + Zd3_A_B[counter2].Lado_B_180Grados;
								ZInternoLastra_A_B[counter2].Lado_B_180Grados := ZCoordinataAppoggioLastra_A_B[counter2].Lado_B_180Grados + (DimensionesPiezasDifEsPiking[counter2].DimPieza_LadoB.YDim / 2) * COS (AngoloAlfa_rad); 	
								
						END_CASE				 
					ELSE
						YCoordinataAppoggioLastra[counter2] := (B/2) + Spessore_Lastra_Inclinata_Cumulato[counter2] + Yd3[counter2];
						YInternoLastra[counter2] := YCoordinataAppoggioLastra[counter2] - (DimensionesPiezasDifEsPiking[counter2].Dim_Horizontal.YDim / 2) * SIN (AngoloAlfa_rad);
						ZCoordinataAppoggioLastra[counter2] := Supporto.ZDim + Zd3[counter2];
						ZInternoLastra[counter2] := ZCoordinataAppoggioLastra[counter2] + (DimensionesPiezasDifEsPiking[counter2].Dim_Horizontal.YDim / 2) * COS (AngoloAlfa_rad); 	
					END_IF
				END_FOR
			END_IF
			
			
	
			(* Calcolo delle coordinate X,Y,Z di ogni singola lastra/falda, centrale o esterno *)
			FOR counter2:=1 TO numeroLastre_int BY 1 DO
				IF  NOT CalculoEstacionPickinPiezasDiferentes  THEN 
					XCentroLastra[counter2] := Supporto.XDim/2;
					YCentroLastra[counter2] := YInternoLastra[counter2] + Yd1[counter2];
					ZCentroLastra[counter2] := ZInternoLastra[counter2] + Zd1[counter2];
					
					XEsternoLastra[counter2] := Supporto.XDim/2;
					YEsternoLastra[counter2] := YInternoLastra[counter2] + Yd2[counter2];	
					ZEsternoLastra[counter2] := ZInternoLastra[counter2] + Zd2[counter2];
				ELSIF CalculoEstacionPickinPiezasDiferentes AND Supporto.Tipologia = CAVALLETTO THEN 
					Fun_PiezaLadoCaballete(Nu_PiezaGlobal:= counter2 , Grados:= ADR(LadoRegistarFor)  ,
										 Nu_pieza_LadoA=>NuPieza_A , Nu_pieza_LadoB=> NuPieza_B  );
					CASE Supporto.TipoTrabajoLado_Cavallete  OF
						0:
							CASE LadoRegistarFor OF
									0: 
										XCentroLastra_A_B[NuPieza_A].Lado_A_0Grados := Supporto.XDim/2;
										YCentroLastra_A_B[NuPieza_A].Lado_A_0Grados := YInternoLastra_A_B[NuPieza_A].Lado_A_0Grados 
																	+ Yd1_A_B[NuPieza_A].Lado_A_0Grados;
										ZCentroLastra_A_B[NuPieza_A].Lado_A_0Grados := ZInternoLastra_A_B[NuPieza_A].Lado_A_0Grados  
																	+	Zd1_A_B[NuPieza_A].Lado_A_0Grados;
										
										XEsternoLastra_A_B[NuPieza_A].Lado_A_0Grados := Supporto.XDim/2;
										YEsternoLastra_A_B[NuPieza_A].Lado_A_0Grados := YInternoLastra_A_B[NuPieza_A].Lado_A_0Grados 
																	+ Yd2_A_B[NuPieza_A].Lado_A_0Grados;	
										ZEsternoLastra_A_B[NuPieza_A].Lado_A_0Grados := ZInternoLastra_A_B[NuPieza_A].Lado_A_0Grados 
																	+ Zd2_A_B[NuPieza_A].Lado_A_0Grados;
								  180:
										XCentroLastra_A_B[NuPieza_B].Lado_B_180Grados := Supporto.XDim/2;
										YCentroLastra_A_B[NuPieza_B].Lado_B_180Grados := YInternoLastra_A_B[NuPieza_B].Lado_B_180Grados 
																	+ Yd1_A_B[NuPieza_B].Lado_B_180Grados;
										ZCentroLastra_A_B[NuPieza_B].Lado_B_180Grados := ZInternoLastra_A_B[NuPieza_B].Lado_B_180Grados 
																	+ Zd1_A_B[NuPieza_B].Lado_B_180Grados;
										
										XEsternoLastra_A_B[NuPieza_B].Lado_B_180Grados := Supporto.XDim/2;
										YEsternoLastra_A_B[NuPieza_B].Lado_B_180Grados := YInternoLastra_A_B[NuPieza_B].Lado_B_180Grados 
																	+ Yd2_A_B[NuPieza_B].Lado_B_180Grados;	
										ZEsternoLastra_A_B[NuPieza_B].Lado_B_180Grados := ZInternoLastra_A_B[NuPieza_B].Lado_B_180Grados 
																	+ Zd2_A_B[NuPieza_B].Lado_B_180Grados;
							END_CASE
						1:
							XCentroLastra_A_B[counter2].Lado_A_0Grados := Supporto.XDim/2;
							YCentroLastra_A_B[counter2].Lado_A_0Grados := YInternoLastra_A_B[counter2].Lado_A_0Grados 
														+ Yd1_A_B[counter2].Lado_A_0Grados;
							ZCentroLastra_A_B[counter2].Lado_A_0Grados := ZInternoLastra_A_B[counter2].Lado_A_0Grados  
														+	Zd1_A_B[counter2].Lado_A_0Grados;
							
							XEsternoLastra_A_B[counter2].Lado_A_0Grados := Supporto.XDim/2;
							YEsternoLastra_A_B[counter2].Lado_A_0Grados := YInternoLastra_A_B[counter2].Lado_A_0Grados 
														+ Yd2_A_B[counter2].Lado_A_0Grados;	
							ZEsternoLastra_A_B[counter2].Lado_A_0Grados := ZInternoLastra_A_B[counter2].Lado_A_0Grados 
														+ Zd2_A_B[counter2].Lado_A_0Grados;
							
						
							
						2:
							XCentroLastra_A_B[counter2].Lado_B_180Grados := Supporto.XDim/2;
							YCentroLastra_A_B[counter2].Lado_B_180Grados := YInternoLastra_A_B[counter2].Lado_B_180Grados 
														+ Yd1_A_B[counter2].Lado_B_180Grados;
							ZCentroLastra_A_B[counter2].Lado_B_180Grados := ZInternoLastra_A_B[counter2].Lado_B_180Grados 
														+ Zd1_A_B[counter2].Lado_B_180Grados;
							
							XEsternoLastra_A_B[counter2].Lado_B_180Grados := Supporto.XDim/2;
							YEsternoLastra_A_B[counter2].Lado_B_180Grados := YInternoLastra_A_B[counter2].Lado_B_180Grados 
														+ Yd2_A_B[counter2].Lado_B_180Grados;	
							ZEsternoLastra_A_B[counter2].Lado_B_180Grados := ZInternoLastra_A_B[counter2].Lado_B_180Grados 
														+ Zd2_A_B[counter2].Lado_B_180Grados;
						
					END_CASE
				ELSIF CalculoEstacionPickinPiezasDiferentes AND Supporto.Tipologia <> CAVALLETTO THEN 
					 
					XCentroLastra[counter2] := Supporto.XDim/2;
					YCentroLastra[counter2] := YInternoLastra[counter2] + Yd1[counter2];
					ZCentroLastra[counter2] := ZInternoLastra[counter2] + Zd1[counter2];
					
					XEsternoLastra[counter2] := Supporto.XDim/2;
					YEsternoLastra[counter2] := YInternoLastra[counter2] + Yd2[counter2];	
					ZEsternoLastra[counter2] := ZInternoLastra[counter2] + Zd2[counter2];
				END_IF
				
			END_FOR;
			
			(* Pulisco le uscite e setto a TERMINATORE tutti gli elementi di FormingSlab*)
			FOR counter1 := 1 TO MAXFORMINGSLAB DO
				FormingSlab.PElement[counter1].Typology := TERMINATORE;
			END_FOR
		//#########################aqui for	
		IF HabiCalTodasCordenadas AND NOT CalculoEstacionPickinPiezasDiferentes THEN
				F_ini := 1 ;
				F_Fin := 4 ;
		ELSIF  CalculoEstacionPickinPiezasDiferentes THEN
				F_ini := TipoOrdinamento ;
				F_Fin := TipoOrdinamento ;
				IF Supporto.TipoTrabajoLado_Cavallete = 0 THEN F_ini := 2 ; F_Fin  := 2 ; END_IF 
				IF Supporto.TipoTrabajoLado_Cavallete = 1 THEN F_ini := 3 ; F_Fin  := 3 ; END_IF 
				IF Supporto.TipoTrabajoLado_Cavallete = 2 THEN F_ini := 4 ; F_Fin  := 4 ; END_IF 
		ELSIF  NOT HabiCalTodasCordenadas AND NOT CalculoEstacionPickinPiezasDiferentes THEN
				F_ini := TipoOrdinamento ;
				F_Fin := TipoOrdinamento ;
				
		END_IF
		
		
		
FOR CalForCavallete := F_ini TO F_Fin DO
	CASE CalForCavallete OF	

				1:	// Lato DX della cavallina
					FOR Contador := 1 TO numeroLastre_int * 2 DO 
						IF NOT 	CalculoEstacionPickinPiezasDiferentes THEN 
							varEven := Contador MOD 2;
								CASE varEven OF
									0:
										XFinale[Contador] := Supporto.XDim/2 + Supporto.OFSDE_X180;
										CASE TipoRisultato OF 
											0:
												XFinale[Contador] := Supporto.XDim/2 + Supporto.OFSDE_X180;
												ZFinale[Contador] := ZInternoLastra[(Contador+varEven)/2] + Supporto.OFSDE_Z180;
											1:
												XFinale[Contador] := Supporto.XDim/2 + Supporto.OFSDE_X180;
												ZFinale[Contador] := ZInternoLastra[(Contador+varEven)/2] + Supporto.OFSDE_Z180;
											3:
												XFinale[Contador] := Supporto.XDim/2 + Supporto.OFSDE_X180;
												ZFinale[Contador] := ZInternoLastra[(Contador+varEven)/2] + Supporto.OFSDE_Z180;
											4:
												XFinale[Contador] := Supporto.XDim/2 + Supporto.OFSDE_X180;
												ZFinale[Contador] := ZInternoLastra[(Contador+varEven)/2] + Supporto.OFSDE_Z180;
										END_CASE
										JFinale[Contador] := 180 - AlgoloAlfa_gradi + Supporto.OFSDE_J180; 
									1: 
										XFinale[Contador] := Supporto.XDim/2 + Supporto.OFSDE_X0;
										CASE TipoRisultato OF 
											1:	
													
													YFinale[Contador] := YInternoLastra[(Contador + varEven)/2] + Supporto.OFSDE_Y0;
													ZFinale[Contador] := ZInternoLastra[(Contador+varEven)/2] 	+ Supporto.OFSDE_Z0;
												2:	
													YFinale[Contador] := YCentroLastra[(Contador + varEven)/2] + Supporto.OFSDE_Y0;
													ZFinale[Contador] := ZCentroLastra[(Contador + varEven)/2] + Supporto.OFSDE_Z0;
												3:	
													YFinale[Contador] := YEsternoLastra[(Contador + varEven)/2] + Supporto.OFSDE_Y0;
													ZFinale[Contador] := ZEsternoLastra[(Contador + varEven)/2] + Supporto.OFSDE_Z0;
												4:	
													YFinale[Contador] := YCoordinataAppoggioLastra[(Contador + varEven)/2] + Supporto.OFSDE_Y0;
													ZFinale[Contador] := ZEsternoLastra[(Contador + varEven)/2] + Supporto.OFSDE_Z0;
											
										END_CASE
										 JFinale[Contador] := AlgoloAlfa_gradi + Supporto.OFSDE_J0;
								END_CASE
						ELSIF CalculoEstacionPickinPiezasDiferentes AND Supporto.Tipologia = CAVALLETTO THEN 
							Fun_PiezaLadoCaballete(Nu_PiezaGlobal:= Contador , Grados:= ADR(LadoRegistarFor)  ,
													 Nu_pieza_LadoA=>NuPieza_A , Nu_pieza_LadoB=> NuPieza_B  );
							CASE TipoRisultato OF 
										1:	
											CASE LadoRegistarFor OF
												0: 
													CoorFinaleLado_Pri0_Des180[NuPieza_A].LadoA.CoordenadaFinale_X := Supporto.XDim/2 + Supporto.OFSDE_X0;;
													CoorFinaleLado_Pri0_Des180[NuPieza_A].LadoA.CoordenadaFinale_Y := YInternoLastra_A_B[NuPieza_A].Lado_A_0Grados + Supporto.OFSDE_Y0;
													CoorFinaleLado_Pri0_Des180[NuPieza_A].LadoA.CoordenadaFinale_Z := ZInternoLastra_A_B[NuPieza_A].Lado_A_0Grados + Supporto.OFSDE_Z0;
													CoorFinaleLado_Pri0_Des180[NuPieza_A].LadoA.CoordenadaFinale_J := AlgoloAlfa_gradi + Supporto.OFSDE_J0 ;
												180 :
													 
													CoorFinaleLado_Pri0_Des180[NuPieza_B].LadoB.CoordenadaFinale_X := Supporto.XDim/2 + Supporto.OFSDE_X180;;
													CoorFinaleLado_Pri0_Des180[NuPieza_B].LadoB.CoordenadaFinale_Y := YInternoLastra_A_B[NuPieza_B].Lado_B_180Grados + Supporto.OFSDE_Y0;
													CoorFinaleLado_Pri0_Des180[NuPieza_B].LadoB.CoordenadaFinale_Z := ZInternoLastra_A_B[NuPieza_B].Lado_B_180Grados + Supporto.OFSDE_Z0;
													CoorFinaleLado_Pri0_Des180[NuPieza_B].LadoB.CoordenadaFinale_J := AlgoloAlfa_gradi + Supporto.OFSDE_J0 ;
											END_CASE
										2:	
											CASE LadoRegistarFor OF
												0: 
													CoorFinaleLado_Pri0_Des180[NuPieza_A].LadoA.CoordenadaFinale_X := Supporto.XDim/2 + Supporto.OFSDE_X0;;
													CoorFinaleLado_Pri0_Des180[NuPieza_A].LadoA.CoordenadaFinale_Y := YCentroLastra_A_B[NuPieza_A].Lado_A_0Grados + Supporto.OFSDE_Y0;
													CoorFinaleLado_Pri0_Des180[NuPieza_A].LadoA.CoordenadaFinale_Z := ZCentroLastra_A_B[NuPieza_A].Lado_A_0Grados + Supporto.OFSDE_Z0;
													CoorFinaleLado_Pri0_Des180[NuPieza_A].LadoA.CoordenadaFinale_J := AlgoloAlfa_gradi + Supporto.OFSDE_J0 ;
												180 :
													 
													CoorFinaleLado_Pri0_Des180[NuPieza_B].LadoB.CoordenadaFinale_X := Supporto.XDim/2 + Supporto.OFSDE_X180;;
													CoorFinaleLado_Pri0_Des180[NuPieza_B].LadoB.CoordenadaFinale_Y := YCentroLastra_A_B[NuPieza_B].Lado_B_180Grados + Supporto.OFSDE_Y0;
													CoorFinaleLado_Pri0_Des180[NuPieza_B].LadoB.CoordenadaFinale_Z := ZCentroLastra_A_B[NuPieza_B].Lado_B_180Grados + Supporto.OFSDE_Z0;
													CoorFinaleLado_Pri0_Des180[NuPieza_B].LadoB.CoordenadaFinale_J := AlgoloAlfa_gradi + Supporto.OFSDE_J0 ;
											END_CASE
										3:	
											CASE LadoRegistarFor OF
												0: 
													CoorFinaleLado_Pri0_Des180[NuPieza_A].LadoA.CoordenadaFinale_X := Supporto.XDim/2 + Supporto.OFSDE_X0;;
													CoorFinaleLado_Pri0_Des180[NuPieza_A].LadoA.CoordenadaFinale_Y := YEsternoLastra_A_B[NuPieza_A].Lado_A_0Grados + Supporto.OFSDE_Y0;
													CoorFinaleLado_Pri0_Des180[NuPieza_A].LadoA.CoordenadaFinale_Z := ZEsternoLastra_A_B[NuPieza_A].Lado_A_0Grados + Supporto.OFSDE_Z0;
													CoorFinaleLado_Pri0_Des180[NuPieza_A].LadoA.CoordenadaFinale_J := AlgoloAlfa_gradi + Supporto.OFSDE_J0 ;
												180 :
													 
